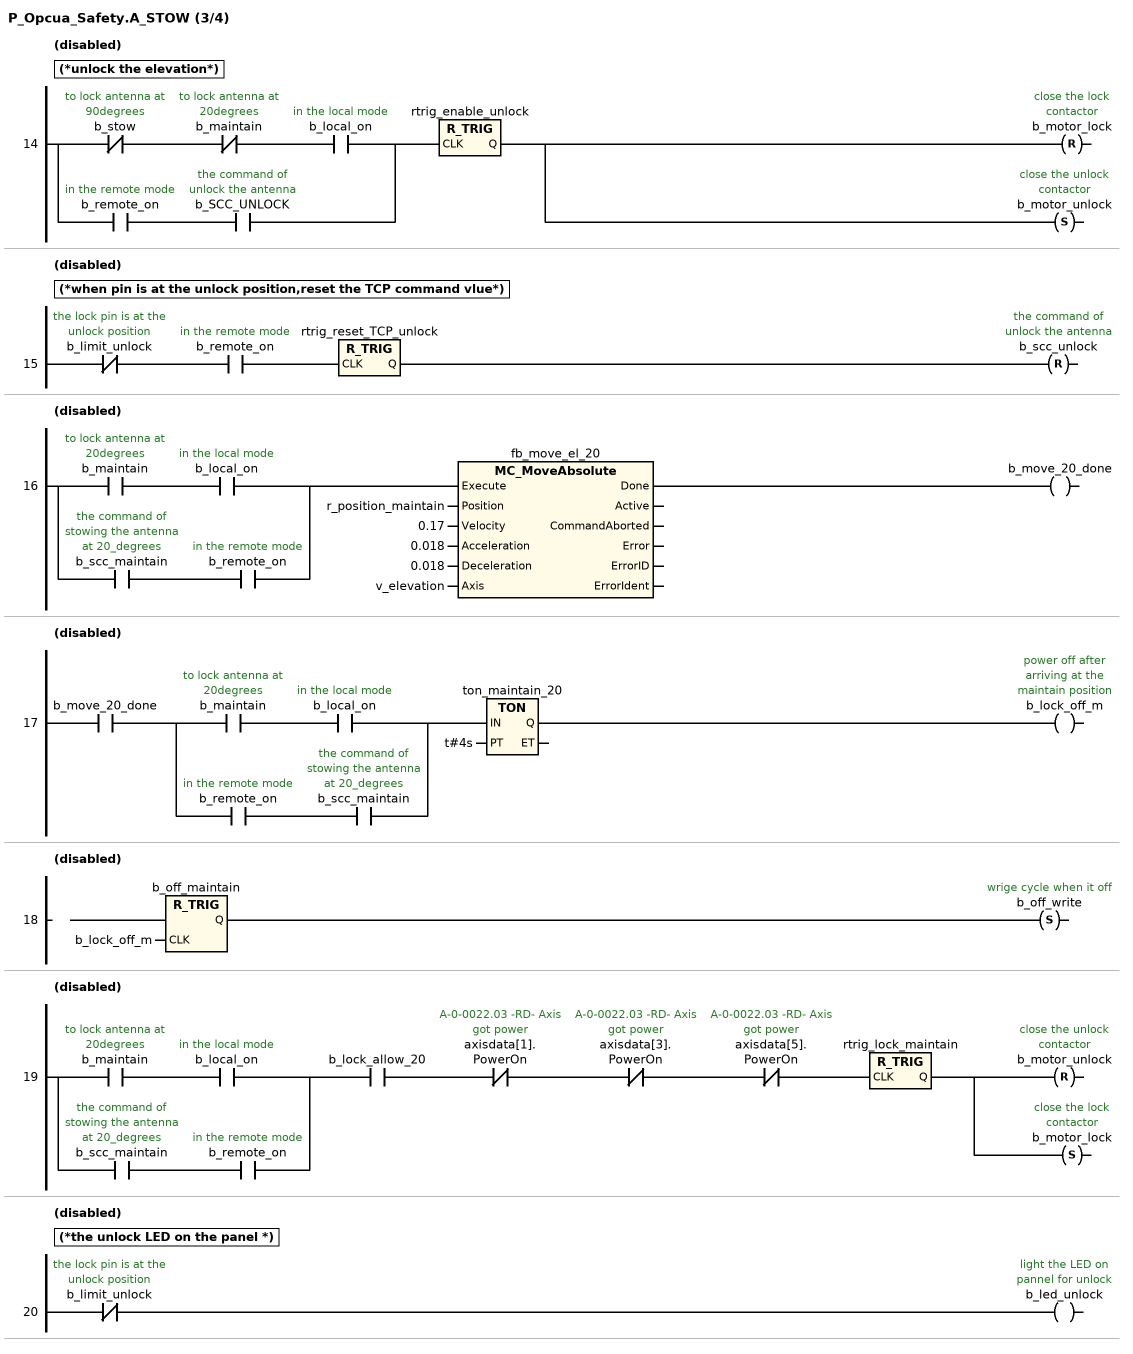
// NETWORK 14 (disabled)
//   b_stow: to lock antenna at 90degrees
//   b_maintain: to lock antenna at 20degrees
//   b_local_on: in the local mode
//   b_remote_on: in the remote mode
//   b_SCC_UNLOCK: the command of unlock the antenna
//   b_motor_lock: close the lock contactor
//   b_motor_unlock: close the unlock contactor
// label: (*unlock the elevation*)
// rtrig_enable_unlock(CLK := NOT b_stow AND NOT b_maintain AND b_local_on OR b_remote_on AND b_SCC_UNLOCK); // R_TRIG
// b_motor_lock R= rtrig_enable_unlock.Q;
// b_motor_unlock S= rtrig_enable_unlock.Q;

// NETWORK 15 (disabled)
//   b_limit_unlock: the lock pin is at the unlock position
//   b_remote_on: in the remote mode
//   b_scc_unlock: the command of unlock the antenna
// label: (*when pin is at the unlock position,reset the TCP command vlue*)
// rtrig_reset_TCP_unlock(CLK := NOT b_limit_unlock AND b_remote_on); // R_TRIG
// b_scc_unlock R= rtrig_reset_TCP_unlock.Q;

// NETWORK 16 (disabled)
//   b_maintain: to lock antenna at 20degrees
//   b_local_on: in the local mode
//   b_scc_maintain: the command of stowing the antenna at 20_degrees
//   b_remote_on: in the remote mode
//   v_elevation: Virtual axis "v_elevation" with axis number 8
// fb_move_el_20(
//     Execute := b_maintain AND b_local_on OR b_scc_maintain AND b_remote_on,
//     Position := r_position_maintain,
//     Velocity := 0.17,
//     Acceleration := 0.018,
//     Deceleration := 0.018,
//     Axis := v_elevation); // MC_MoveAbsolute
// b_move_20_done := fb_move_el_20.Done;

// NETWORK 17 (disabled)
//   b_maintain: to lock antenna at 20degrees
//   b_local_on: in the local mode
//   b_remote_on: in the remote mode
//   b_scc_maintain: the command of stowing the antenna at 20_degrees
//   b_lock_off_m: power off after arriving at the maintain position
// ton_maintain_20(IN := b_move_20_done AND (b_maintain AND b_local_on OR b_remote_on AND b_scc_maintain), PT := t#4s); // TON
// b_lock_off_m := ton_maintain_20.Q;

// NETWORK 18 (disabled)
//   b_lock_off_m: power off after arriving at the maintain position
//   b_off_write: wrige cycle when it off
// b_off_maintain(CLK := b_lock_off_m); // R_TRIG
// b_off_write S= b_off_maintain.Q;

// NETWORK 19 (disabled)
//   b_maintain: to lock antenna at 20degrees
//   b_local_on: in the local mode
//   b_scc_maintain: the command of stowing the antenna at 20_degrees
//   b_remote_on: in the remote mode
//   axisdata[1].PowerOn: A-0-0022.03 -RD- Axis got power
//   axisdata[3].PowerOn: A-0-0022.03 -RD- Axis got power
//   axisdata[5].PowerOn: A-0-0022.03 -RD- Axis got power
//   b_motor_unlock: close the unlock contactor
//   b_motor_lock: close the lock contactor
// rtrig_lock_maintain(CLK := (b_maintain AND b_local_on OR b_scc_maintain AND b_remote_on) AND b_lock_allow_20 AND NOT axisdata[1].PowerOn AND NOT axisdata[3].PowerOn AND NOT axisdata[5].PowerOn); // R_TRIG
// b_motor_unlock R= rtrig_lock_maintain.Q;
// b_motor_lock S= rtrig_lock_maintain.Q;

// NETWORK 20 (disabled)
//   b_limit_unlock: the lock pin is at the unlock position
//   b_led_unlock: light the LED on pannel for unlock
// label: (*the unlock LED on the panel *)
// b_led_unlock := NOT b_limit_unlock;

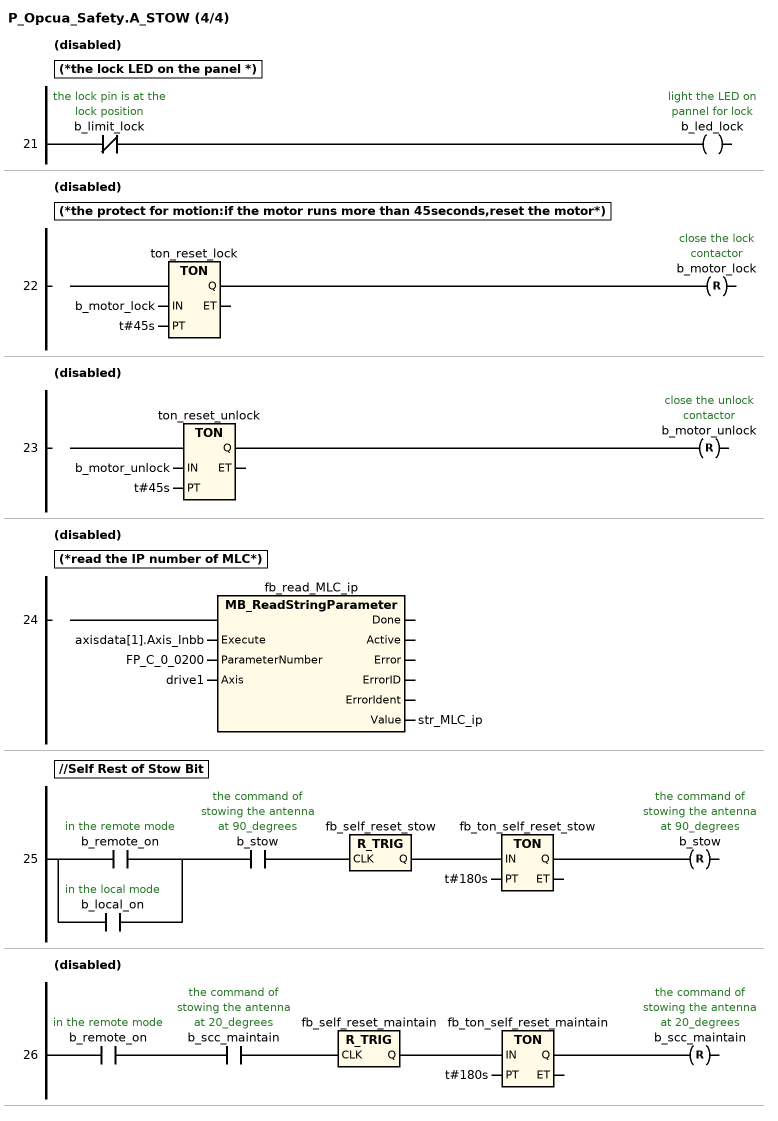
// NETWORK 21 (disabled)
//   b_limit_lock: the lock pin is at the lock position
//   b_led_lock: light the LED on pannel for lock
// label: (*the lock LED on the panel *)
// b_led_lock := NOT b_limit_lock;

// NETWORK 22 (disabled)
//   b_motor_lock: close the lock contactor
// label: (*the protect for motion:if the motor runs more than 45seconds,reset the motor*)
// ton_reset_lock(IN := b_motor_lock, PT := t#45s); // TON
// b_motor_lock R= ton_reset_lock.Q;

// NETWORK 23 (disabled)
//   b_motor_unlock: close the unlock contactor
// ton_reset_unlock(IN := b_motor_unlock, PT := t#45s); // TON
// b_motor_unlock R= ton_reset_unlock.Q;

// NETWORK 24 (disabled)
//   axisdata[1].Axis_Inbb: A-0-0021.13 -RD- Axis is ready for power to the amplifier (bb)
//   FP_C_0_0200: Engineering, IP address
//   drive1: Real axis "Drive1" with axis number 1
//   str_MLC_ip: IP number in MLC
// label: (*read the IP number of MLC*)
// fb_read_MLC_ip(
//     Execute := axisdata[1].Axis_Inbb,
//     ParameterNumber := FP_C_0_0200,
//     Axis := drive1,
//     Value => str_MLC_ip); // MB_ReadStringParameter

// NETWORK 25
//   b_remote_on: in the remote mode
//   b_local_on: in the local mode
//   b_stow: the command of stowing the antenna at 90_degrees
// label: //Self Rest of Stow Bit
fb_self_reset_stow(CLK := (b_remote_on OR b_local_on) AND b_stow); // R_TRIG
fb_ton_self_reset_stow(IN := fb_self_reset_stow.Q, PT := t#180s); // TON
b_stow R= fb_ton_self_reset_stow.Q;

// NETWORK 26 (disabled)
//   b_remote_on: in the remote mode
//   b_scc_maintain: the command of stowing the antenna at 20_degrees
// fb_self_reset_maintain(CLK := b_remote_on AND b_scc_maintain); // R_TRIG
// fb_ton_self_reset_maintain(IN := fb_self_reset_maintain.Q, PT := t#180s); // TON
// b_scc_maintain R= fb_ton_self_reset_maintain.Q;
END_ACTION

ACTION A_Interlock_Estop:
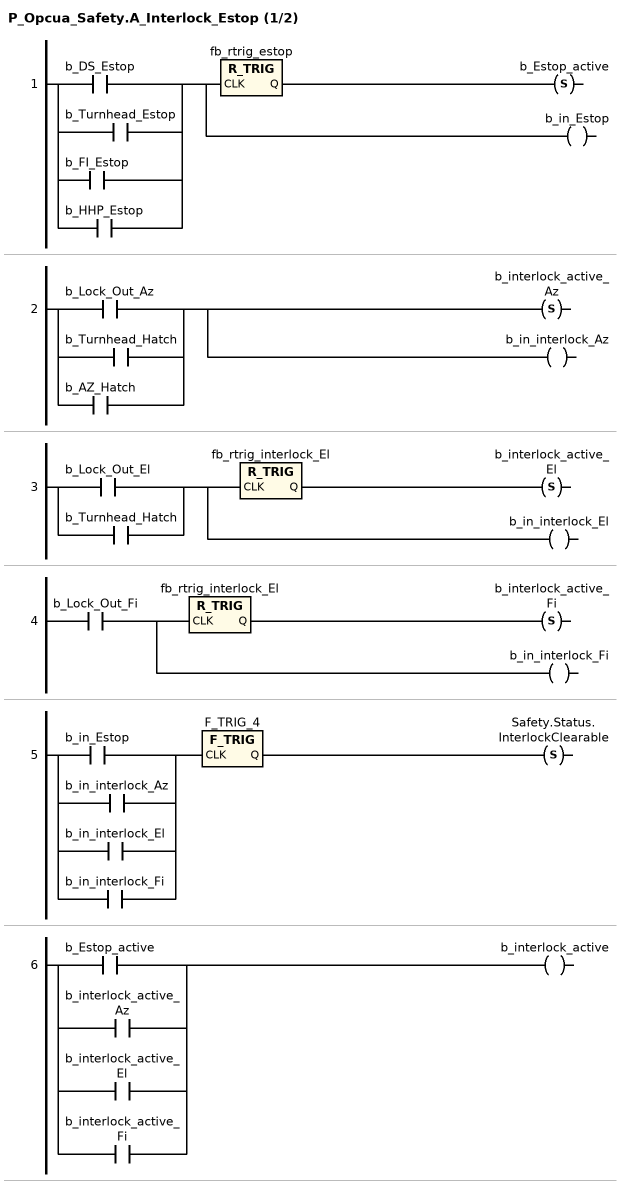
// NETWORK 1
_w3 := b_DS_Estop OR b_Turnhead_Estop OR b_FI_Estop OR b_HHP_Estop;
fb_rtrig_estop(CLK := _w3); // R_TRIG
b_Estop_active S= fb_rtrig_estop.Q;
b_in_Estop := _w3;

// NETWORK 2
_w4 := b_Lock_Out_Az OR b_Turnhead_Hatch OR b_AZ_Hatch;
b_interlock_active_Az S= _w4;
b_in_interlock_Az := _w4;

// NETWORK 3
_w5 := b_Lock_Out_El OR b_Turnhead_Hatch;
fb_rtrig_interlock_El(CLK := _w5); // R_TRIG
b_interlock_active_El S= fb_rtrig_interlock_El.Q;
b_in_interlock_El := _w5;

// NETWORK 4
fb_rtrig_interlock_El(CLK := b_Lock_Out_Fi); // R_TRIG
b_interlock_active_Fi S= fb_rtrig_interlock_El.Q;
b_in_interlock_Fi := b_Lock_Out_Fi;

// NETWORK 5
F_TRIG_4(CLK := b_in_Estop OR b_in_interlock_Az OR b_in_interlock_El OR b_in_interlock_Fi); // F_TRIG
Safety.Status.InterlockClearable S= F_TRIG_4.Q;

// NETWORK 6
b_interlock_active := b_Estop_active OR b_interlock_active_Az OR b_interlock_active_El OR b_interlock_active_Fi;

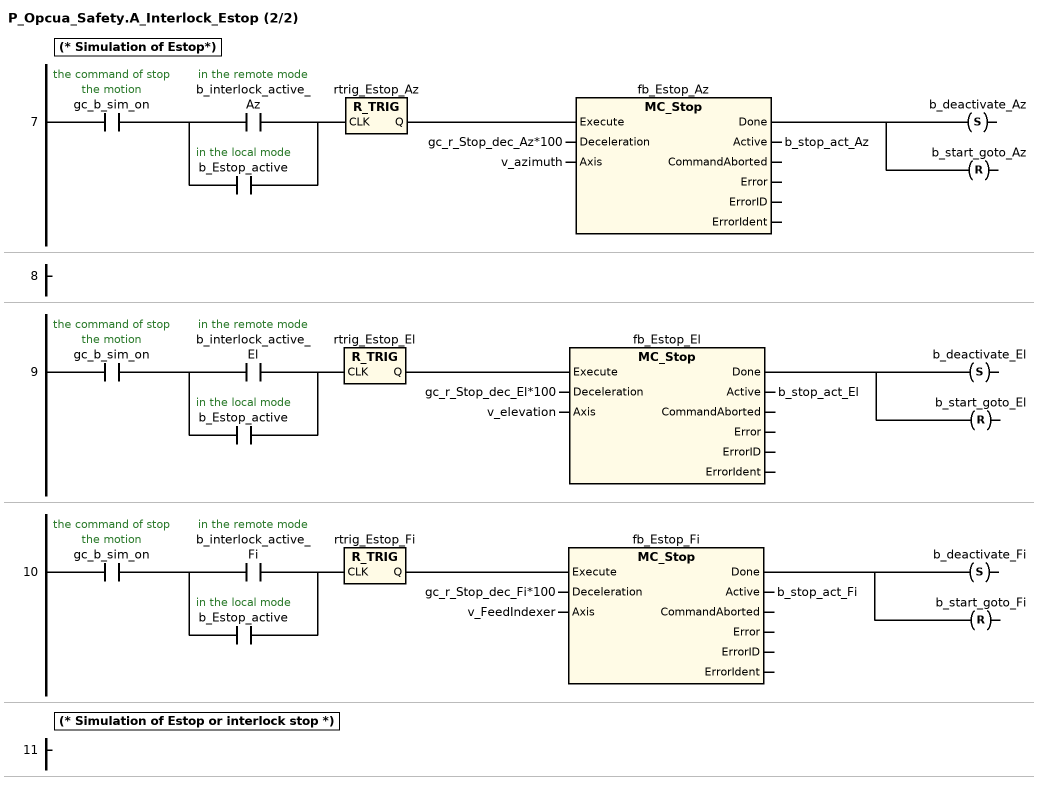
// NETWORK 7
//   gc_b_sim_on: the command of stop the motion
//   b_interlock_active_Az: in the remote mode
//   b_Estop_active: in the local mode
//   v_azimuth: Virtual axis "v_azimuth" with axis number 7
// label: (* Simulation of Estop*)
rtrig_Estop_Az(CLK := gc_b_sim_on AND (b_interlock_active_Az OR b_Estop_active)); // R_TRIG
fb_Estop_Az(
    Execute := rtrig_Estop_Az.Q,
    Deceleration := gc_r_Stop_dec_Az*100,
    Axis := v_azimuth,
    Active => b_stop_act_Az); // MC_Stop
b_deactivate_Az S= fb_Estop_Az.Done;
b_start_goto_Az R= fb_Estop_Az.Done;

// NETWORK 8

// NETWORK 9
//   gc_b_sim_on: the command of stop the motion
//   b_interlock_active_El: in the remote mode
//   b_Estop_active: in the local mode
//   v_elevation: Virtual axis "v_elevation" with axis number 8
rtrig_Estop_El(CLK := gc_b_sim_on AND (b_interlock_active_El OR b_Estop_active)); // R_TRIG
fb_Estop_El(
    Execute := rtrig_Estop_El.Q,
    Deceleration := gc_r_Stop_dec_El*100,
    Axis := v_elevation,
    Active => b_stop_act_El); // MC_Stop
b_deactivate_El S= fb_Estop_El.Done;
b_start_goto_El R= fb_Estop_El.Done;

// NETWORK 10
//   gc_b_sim_on: the command of stop the motion
//   b_interlock_active_Fi: in the remote mode
//   b_Estop_active: in the local mode
//   v_FeedIndexer: Virtual axis "v_polarization" with axis number 9
rtrig_Estop_Fi(CLK := gc_b_sim_on AND (b_interlock_active_Fi OR b_Estop_active)); // R_TRIG
fb_Estop_Fi(
    Execute := rtrig_Estop_Fi.Q,
    Deceleration := gc_r_Stop_dec_Fi*100,
    Axis := v_FeedIndexer,
    Active => b_stop_act_Fi); // MC_Stop
b_deactivate_Fi S= fb_Estop_Fi.Done;
b_start_goto_Fi R= fb_Estop_Fi.Done;

// NETWORK 11
// label: (* Simulation of Estop or interlock stop *)
END_ACTION

END_PROGRAM

// IndraMotionMlc1/Application/POUs/OPCUA/OPCUA_Node/P_Opcua_CommandArbiter
PROGRAM P_Opcua_CommandArbiter
VAR
	cmds: CmdResponseType;
END_VAR

CommandArbiter();
//CommandArbiter.Status.DscCmdAuthority;


(* if hhp connected then 
    CommandArbiter.DscCmdAuthority:= HHP;
	End *)

END_PROGRAM

// IndraMotionMlc1/Application/POUs/OPCUA/OPCUA_Node/P_Opcua_Time_cds
PROGRAM P_Opcua_Time_cds
VAR
	IL_SysTime64_0: IL_SysTime64;
	Current_time: SYS_TIME64;
	UnixSeconds: Lreal;
	i_num_quarter_test: DINT;
	current_time_pos_test: LREAL;
	lr_MJD_Test: LREAL;
	
	dummy: Lreal;
	dummy2: Bool;
END_VAR

Time_cds();

P_Opcua_Time_cds.Get_Time();
//Time_cds.Status.TAIOffset:=Current_time.HighValue*65536+Current_time.LowValue;
//Calculate TAI offset 
//Time_cds.Status.TAIOffset:=Current_time.HighValue*65536+Current_time.LowValue;
//Time_cds.Status.TAIOffset:=((Current_time.HighValue+4294967295)/1000000+ Current_time.LowValue/1000000);
UnixSeconds:=(TO_LREAL(Current_time.HighValue)*4294967295+TO_LREAL(Current_time.LowValue))/1000000; //UTC 
//Time_cds.Status.TAIOffset:=UnixSeconds-UnixToSKAEpoch-(Time_cds.Status.LeapSecPTP-Time_cds.Status.UTCtoSkaoEpochSec);

lr_MJD_Test:= UnixSeconds/86400+40587;

 // This should be the TAI offset after the SKAO epoch. The time from the Time Virtual axis.
//Time_cds.Status.DscTimeSyncSource:=Source_Timesync;

Time_cds.Status.LeapSecPTP:=LeapSecPTP;   
IF Source_Timesync = DscTimeSyncSourceType.PTP THEN
	Time_cds.Status.TimeSourceAddrNTP:=IP_Adress_PTP;
ELSIF Source_Timesync = DscTimeSyncSourceType.NTP THEN
	Time_cds.Status.TimeSourceAddrNTP:=IP_Adress_NTP;
ELSE
	Time_cds.Status.TimeSourceAddrNTP:=str_MLC_ip;
END_IF

IF Source_Timesync = DscTimeSyncSourceType.PTP THEN
	Time_cds.Status.TimeSynced:=b_M_time_done;
	b_no_SetDateTime:=FALSE;
ELSIF Source_Timesync = DscTimeSyncSourceType.NTP THEN
	//Time_cds.Status.TimeSynced:=b_M_time_done;
	b_no_SetDateTime:=FALSE;
ELSE
	
    Time_cds.Status.TimeSynced:=b_M_time_done;
	// need to use system time to calculate MJD
	b_no_SetDateTime:=TRUE;
	
	di_MJD_day := LREAL_TO_DINT(TRUNC(UnixSeconds/86400+40587));
	i_num_quarter:=TRUNC((UnixSeconds-DINT_TO_LREAL(TRUNC(UnixSeconds/86400)*86400))/360);
	current_time_pos_test:=UnixSeconds-DINT_TO_LREAL(TRUNC(UnixSeconds/86400)*86400)-i_num_quarter*360;
	dummy:=P_UDP_To_NTP.current_time_pos-current_time_pos_test;
	dummy2:=(ABS(dummy)>=0.10);
	IF (ABS(dummy)>=0.10 AND NOT(b_track_on)) THEN
		P_UDP_To_NTP.current_time_pos:=current_time_pos_test;
	   	P_UDP_To_NTP.b_NTP_set_up:=TRUE;
	ELSE 
		P_UDP_To_NTP.b_NTP_set_up:=FALSE;	
	
	END_IF
	
	
	
END_IF

ACTION Get_Time:
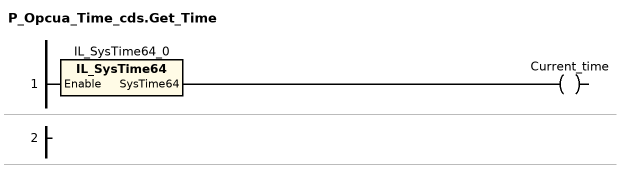
// NETWORK 1
IL_SysTime64_0(Enable := TRUE); // IL_SysTime64
Current_time := IL_SysTime64_0.SysTime64;

// NETWORK 2
END_ACTION

END_PROGRAM

// IndraMotionMlc1/Application/POUs/OPCUA/OPCUA_Node/P_Opcua_Management
PROGRAM P_Opcua_Management
VAR
	R_total_distance_AZ_old:LREAL;
	R_total_distance_EL_deg_old:LREAL;
	R_total_distance_EL_m_old:LREAL;
	R_total_distance_FI_old:LREAL;
	count_i:UINT;
	(*<<<<<<<<<<<<<<<<<<<<<<<<<<<<<<<<<<<< Stop >>>>>>>>>>>>>>>>>>>>>>>>>>>>>*)
	b_stop_Az_done: BOOL;
	b_stop_El_done: BOOL;
	b_stop_Fi_done: BOOL;
	fb_stop_Az: MC_Stop;
	fb_stop_El: MC_Stop;
	fb_stop_Fi: MC_Stop;
	rtrig_stop_Az: R_TRIG;
	rtrig_stop_El: R_TRIG;
	rtrig_stop_Fi: R_TRIG;
	rtrig_stop_stow: R_TRIG;
	rtrig_reset_stop: R_TRIG;
	
	(*<<<<<<<<<<<<<<<<<<<<<<<<<<<<<<<<<<<< Goto >>>>>>>>>>>>>>>>>>>>>>>>>>>>>*)
	// Az
	
	b_goto_done_Az: BOOL;
	b_active_Az:     BOOL;
	b_moving_Az: BOOL;
	fb_goto_Az: MC_MoveRelative;
	fb_start_goto_Az: R_Trig;
	fb_goto_done_Az : R_Trig;
	
	// El
	
	b_goto_done_El: BOOL;
	b_active_El:     BOOL;
	b_moving_El: BOOL;
	fb_goto_El: MC_MoveRelative;
	fb_start_goto_El: R_Trig;
	fb_goto_done_El : R_Trig;
	//Fi
	b_goto_done_Fi: BOOL;
	b_active_Fi:     BOOL;
	b_moving_Fi: BOOL;
	fb_goto_Fi: MC_MoveRelative;
	fb_start_goto_Fi: R_Trig;
	fb_goto_done_Fi : R_Trig;
	
(*<<<<<<<<<<<<<<<<<<<<<<<<<<<<<<<<<<<<<<<<<<<<<<<<<<<power>>>>>>>>>>>>>>>>>>>>>>>>>>>>>>>>>>>>*)
	ton_pow_off_Az: TON;
	ton_pow_off_El: TON;
	ton_pow_off_Fi: TON;
	rtrig_power_Az: R_TRIG;
	rtrig_power_El: R_TRIG;
	rtrig_power_Fi: R_TRIG;
	fb_ton_El: TON;
	fb_ton_Fi: TON;
	rtrig_off_Az: R_TRIG;
	rtrig_off_El: R_TRIG;
	rtrig_off_Fi: R_TRIG;
	rtrig_power_power: R_TRIG;
	b_pwr_on:BOOL;
	b_pwr_off: BOOL;
	b_clear_off_done_Az1: BOOL;
	b_clear_off_done_Az2: BOOL;
	b_clear_off_done_El: BOOL;
	b_clear_off_done_Fi1: BOOL;
	b_clear_off_done_Fi2: BOOL;
	
	FB_clear_error_off_Az1:MB_WriteParameter;
	FB_clear_error_off_Az2:MB_WriteParameter;
	FB_clear_error_off_El:MB_WriteParameter;
	FB_clear_error_off_Fi1:MB_WriteParameter;
	FB_clear_error_off_Fi2:MB_WriteParameter;
	rtrig_err: R_TRIG;
	rtrig_clear_done: R_TRIG;
	fb_ton_stow: TON;
	
	fb_rtrig_stow_deactivate1: R_TRIG;
	fb_rtrig_stow_deactivate: R_TRIG;
	b_execute_goto_Az: BOOL;
	TON_0: TON;
	R_TRIG_0: R_TRIG;
	R_TRIG_1: R_TRIG;
	TON_1: TON;
END_VAR


(***********Management.DscState***********)
IF azimuth.Status.AxisState=axisstatetype.StartUp OR elevation.Status.AxisState=axisstatetype.StartUp THEN
	Management.Status.DscState:=DscstateType.StartUp;
END_IF

IF azimuth.Status.AxisState=axisstatetype.Standby AND elevation.Status.AxisState=axisstatetype.Standby THEN
	Management.Status.DscState:=DscstateType.Standby;
END_IF

IF azimuth.Status.AxisState=axisstatetype.Activating OR elevation.Status.AxisState=axisstatetype.Activating THEN
	Management.Status.DscState:=DscstateType.Activating;
END_IF

IF azimuth.Status.AxisState=axisstatetype.Deactivating OR elevation.Status.AxisState=axisstatetype.Deactivating THEN
	Management.Status.DscState:=DscstateType.Deactivating;
END_IF

IF azimuth.Status.AxisState=axisstatetype.Standstill OR elevation.Status.AxisState=axisstatetype.Standstill THEN
	Management.Status.DscState:=DscstateType.Standstill;
END_IF

IF azimuth.Status.AxisState=axisstatetype.Stopping OR elevation.Status.AxisState=axisstatetype.Stopping THEN
	Management.Status.DscState:=DscstateType.stopping;
END_IF

IF azimuth.Status.AxisState=axisstatetype.Jog OR elevation.Status.AxisState=axisstatetype.Jog THEN
	Management.Status.DscState:=DscstateType.Jog;
END_IF

IF azimuth.Status.AxisState=axisstatetype.Slew OR elevation.Status.AxisState=axisstatetype.Slew THEN //capitalise S in slew
	Management.Status.DscState:=DscstateType.slew;
END_IF

IF azimuth.Status.AxisState=axisstatetype.Track AND elevation.Status.AxisState=axisstatetype.Track THEN
	Management.Status.DscState:=DscstateType.Track;
END_IF

IF azimuth.Status.AxisState=axisstatetype.Stowed THEN
	Management.Status.DscState:=DscstateType.Stowed;
END_IF
IF azimuth.Status.AxisState=axisstatetype.Locked OR elevation.Status.AxisState=axisstatetype.Locked THEN
	Management.Status.DscState:=DscstateType.Locked;
END_IF

IF azimuth.Status.AxisState=axisstatetype.Locked_Stowed OR elevation.Status.AxisState=axisstatetype.Locked_Stowed THEN
	Management.Status.DscState:=DscstateType.Locked_Stowed;
END_IF

// This one isn't going to work 
IF b_stow_pin_limit_lock AND (azimuth.Status.AxisState=axisstatetype.Locked OR elevation.Status.AxisState=axisstatetype.Locked) THEN     // Need to check Errors and interlocks to go into locked
	Management.Status.DscState:=DscstateType.Locked_Stowed;
END_IF

(*IF b_in_Estop THEN
	Management.Status.DscState:=DscstateType.Locked;  //Axis also need to go into locked state
END_IF
*)


// Work out where FiPOS is 
IF b_goto_done_Fi THEN 
	IF r_pos_fi_v < gc_r_band_optical+gc_r_band_tolerance AND r_pos_fi_v > gc_r_band_optical-gc_r_band_tolerance THEN 
		Management.Status.FiPos:= bandtype.Optical;
	ELSIF
		r_pos_fi_v < gc_r_band_1+gc_r_band_tolerance AND r_pos_fi_v > gc_r_band_1-gc_r_band_tolerance THEN 
		Management.Status.FiPos:= bandtype.Band_1;
	ELSIF
		r_pos_fi_v < gc_r_band_2+gc_r_band_tolerance AND r_pos_fi_v > gc_r_band_2-gc_r_band_tolerance THEN 
		Management.Status.FiPos:= bandtype.Band_2;
	ELSIF
		r_pos_fi_v < gc_r_band_3+gc_r_band_tolerance AND r_pos_fi_v > gc_r_band_3-gc_r_band_tolerance THEN 
		Management.Status.FiPos:= bandtype.Band_3;
	ELSIF
		r_pos_fi_v < gc_r_band_4+gc_r_band_tolerance AND r_pos_fi_v > gc_r_band_4-gc_r_band_tolerance THEN 
		Management.Status.FiPos:= bandtype.Band_4;
	ELSIF
		r_pos_fi_v < gc_r_band_5a+gc_r_band_tolerance AND r_pos_fi_v > gc_r_band_5a-gc_r_band_tolerance THEN 
		Management.Status.FiPos:= bandtype.Band_5a;
	ELSIF
		r_pos_fi_v < gc_r_band_5b+gc_r_band_tolerance AND r_pos_fi_v > gc_r_band_5b-gc_r_band_tolerance THEN 
		Management.Status.FiPos:= bandtype.Band_5b;
	ELSIF
		r_pos_fi_v < gc_r_band_6+gc_r_band_tolerance AND r_pos_fi_v > gc_r_band_6-gc_r_band_tolerance THEN 
		Management.Status.FiPos:= bandtype.Band_6;
	ELSE
		Management.Status.FiPos:= bandtype.Unknown;
	END_IF

END_IF


//Management.Status.FiPos:=Current_FIPos; // this needs to be of band type 
Management.Status.HHP_Cncted:=b_HHP_Connected;
Management.Status.HHP_Az:=b_HHP_AZ;
Management.Status.HHP_El:=b_HHP_EL;
IF b_HHP_AZ = FALSE AND b_HHP_EL= FALSE THEN
	Management.Status.HHP_Fi:=TRUE;
ELSE
	Management.Status.HHP_Fi:=FALSE;
END_IF
IF b_HHP_move_cw_slow OR b_HHP_move_cw_fast THEN
	Management.Status.HHP_Dir_Plus	:= TRUE;
ELSE
	Management.Status.HHP_Dir_Plus	:= FALSE;
END_IF
IF b_HHP_move_ccw_slow OR b_HHP_move_ccw_fast THEN
	Management.Status.HHP_Dir_Minus:= TRUE;
ELSE
	Management.Status.HHP_Dir_Minus:= FALSE;
END_IF

(*********NamePlate**********)
Management.NamePlate.RunHours:=r_operation_hour;

count_i:=count_i+1;
IF count_i = 5 THEN
	R_total_distance_AZ:=ABS(r_pos_az-R_total_distance_AZ_old)+R_total_distance_AZ;
	R_total_distance_AZ_old:=r_pos_az;
	R_total_distance_EL_deg:=ABS(r_pos_el-R_total_distance_el_deg_old)+R_total_distance_el_deg;
	R_total_distance_EL_m:=R_total_distance_EL_deg/K_gear_ratio;
	R_total_distance_el_deg_old:=r_pos_el;
	R_total_distance_FI:=ABS(r_pos_FI-R_total_distance_FI_old)+R_total_distance_FI;
	R_total_distance_FI_old:=r_pos_FI;
	count_i:=0;
END_IF

Management.NamePlate.TotalDist_Az:=R_total_distance_AZ;
Management.NamePlate.TotalDist_El_deg:=R_total_distance_EL_deg;
Management.NamePlate.TotalDist_El_m:=R_total_distance_EL_m;
Management.NamePlate.TotalDist_Fi:=R_total_distance_FI;

(*********TempHumidStatus**********)
Management.TempHumidStatus.HumidDriveCab:=LREAL_TO_REAL(HumidDriveCab);
Management.TempHumidStatus.TempDriveCab:=LREAL_TO_REAL(TempDriveCab);
Management.TempHumidStatus.HumidPSC_Inlet:=LREAL_TO_REAL(HumidPSC_Inlet);
Management.TempHumidStatus.TempPSC_Inlet:=LREAL_TO_REAL(TempPSC_Inlet);
Management.TempHumidStatus.HumidPSC_Outlet:=LREAL_TO_REAL(HumidPSC_Outlet);
Management.TempHumidStatus.TempPSC_Outlet:=LREAL_TO_REAL(TempPSC_Outlet);
Management.TempHumidStatus.TempEMISC_Outlet:=LREAL_TO_REAL(TempEMISC_Outlet);

(*********PowerStatus**********)
Management.PowerStatus.cbEMISC:=b_PSC_PD_EMISC_Breaker_on;
Management.PowerStatus.cbFan_PSC:=b_PSC_PD_FAN_Breaker_on;
Management.PowerStatus.cbPSC_Spare:=b_PSC_PD_spare;
Management.PowerStatus.cbHe_Comp:=b_MAIN_PD_Compressor_breaker_on;
Management.PowerStatus.cbPDU_Fi:=b_MAIN_PD_FI_Breaker_on;
Management.PowerStatus.cbPED_Spare:=b_MAIN_PD_spare;
Management.PowerStatus.ActPwrCnsm:= 0; // Needs to be updated with real number
Management.PowerStatus.CurrentPh1:= LREAL_TO_REAL(CurrentPh1);
Management.PowerStatus.CurrentPh2:=LREAL_TO_REAL(CurrentPh2);
Management.PowerStatus.CurrentPh3:=LREAL_TO_REAL(CurrentPh3);
Management.PowerStatus.FrequencyPh1:=LREAL_TO_REAL(FrequencyPh1);
Management.PowerStatus.FrequencyPh2:=LREAL_TO_REAL(FrequencyPh2);
Management.PowerStatus.FrequencyPh3:=LREAL_TO_REAL(FrequencyPh3);
Management.PowerStatus.VoltagePh1:=LREAL_TO_REAL(VoltagePh1);
Management.PowerStatus.VoltagePh2:=LREAL_TO_REAL(VoltagePh2);
Management.PowerStatus.VoltagePh3:=LREAL_TO_REAL(VoltagePh3);
Management.PowerStatus.PowerFactor:=LREAL_TO_REAL(PowerFactor);
//Management.PowerStatus.LowPowerActive:=0;  

(*********ErrorStatus**********)

//Management.ErrorStatus.errAuthLost:=0;
Management.ErrorStatus.errAzimuth:=(axisdata[1].Axis_Error OR axisdata[2].Axis_Error);  
Management.ErrorStatus.errElevation:=(axisdata[3].Axis_Error);  
Management.ErrorStatus.errFeedindexer:=(axisdata[4].Axis_Error OR axisdata[5].Axis_Error); 
Management.ErrorStatus.errPoint:=0;
IF safety.Status.SafetyState=0 THEN
	Management.ErrorStatus.errSafety:=0;
ELSE
	Management.ErrorStatus.errSafety:=1;
END_IF
Management.ErrorStatus.errTime:=axisdata[10].Axis_Error;
Management.ErrorStatus.errCmd:=Command_Arbiter_error;
Management.ErrorStatus.errTrack:=(NOT(tracking.Status.tr_initOk) AND b_track_on);
Management.ErrorStatus.errStwPin:=NOT((b_stow_pin_limit_lock XOR b_stow_pin_limit_unlock)XOR(b_stow_pin_retract XOR b_stow_pin_deploy));
IF status_code1 = 'F8070' OR status_code2 = 'F8070' OR status_code3 = 'F8070' OR status_code4 = 'F8070' OR status_code5 = 'F8070' THEN
	Management.ErrorStatus.errPwr24VDC:=1;
ELSE
	Management.ErrorStatus.errPwr24VDC:=0;
END_IF
IF status_code1 = 'F2802' OR status_code2 = 'F2802' OR status_code3 = 'F2802' OR status_code4 = 'F2802' OR status_code5 = 'F2802' THEN
	Management.ErrorStatus.errPwr400VAC:=1;
ELSE
	Management.ErrorStatus.errPwr400VAC:=0;
END_IF
IF status_code1 = 'F2802' OR status_code2 = 'F2802' OR status_code3 = 'F2802' OR status_code4 = 'F2802' OR status_code5 = 'F2802' THEN
	Management.ErrorStatus.errPwr400VAC:=1;
ELSE
	Management.ErrorStatus.errPwr400VAC:=0;
END_IF
IF status_code1 = 'F8091' OR status_code2 = 'F8091' OR status_code3 = 'F8091' OR status_code4 = 'F8091' OR status_code5 = 'F8091' THEN
	Management.ErrorStatus.errPwr400VAC:=1;
ELSE
	Management.ErrorStatus.errPwr400VAC:=0;
END_IF
//	Management.ErrorStatus.errPwrMeterComms:=0;
//	Management.ErrorStatus.errTiltOneComms:=0;
//	Management.ErrorStatus.errTiltOneIoUnit:=0;
//	Management.ErrorStatus.errTiltTwoComms:=0;
//	Management.ErrorStatus.errTiltTwoIoUnit:=0;

Management.ErrorStatus.errGeneral:=(Management.ErrorStatus.errAzimuth OR Management.ErrorStatus.errElevation OR Management.ErrorStatus.errFeedindexer OR Management.ErrorStatus.errSafety OR Management.ErrorStatus.errTime OR Management.ErrorStatus.errTrack OR Management.ErrorStatus.errPoint);
Management.ErrorStatus.errMngmnt:=Management.ErrorStatus.errGeneral;

(*********WarningStatus**********)
//IF gc_b_sim_on = 0 THEN 
	Management.WarningStatus.waAzimuth:=(axisdata[1].Axis_Warning OR axisdata[2].Axis_Warning);
    Management.WarningStatus.waElevation:=(axisdata[3].Axis_Warning);
    Management.WarningStatus.waFeedindexer:=(axisdata[4].Axis_Warning OR axisdata[5].Axis_Warning);
//ELSIF gc_b_sim_on =1 THEN
//	Management.WarningStatus.waAzimuth:=(

Management.WarningStatus.waCmd:=0;
Management.WarningStatus.waPoint:=0;
Management.WarningStatus.waSafety:=0;
Management.WarningStatus.waStwPin:=0;
Management.WarningStatus.waPoint:=0;
Management.WarningStatus.waTime:=0;
Management.WarningStatus.waTrack:=0;
Management.WarningStatus.waDoorDrive:=b_DriveCabinetDoor_Estop;
Management.WarningStatus.waDoorEMISC:=b_EMISCDoor_Estop;
Management.WarningStatus.waDoorPED:=b_DSDoor_Estop;
Management.WarningStatus.waDoorPSC:=b_PSCDoor_Estop;
Management.WarningStatus.waHatchPscRoof:=0;
Management.WarningStatus.waHatchAzBearing:=b_AZ_Hatch;
Management.WarningStatus.waHornOn:=b_Horn;
//Management.WarningStatus.waOverTempDrive
//Management.WarningStatus.waOverTempEMISC
//Management.WarningStatus.waDoorPED
//Management.WarningStatus.waDoorPSC
Management.WarningStatus.waSafe2ApproachLight:=0;

// Power mode control 
// Need to limit velocity and acceleration to keep the power below the limit 


// Run Ladder logic
P_Opcua_Management.A_CLR_ERR();
P_Opcua_Management.A_STOP();
P_Opcua_Management.A_GOTO();

ACTION A_STOP:
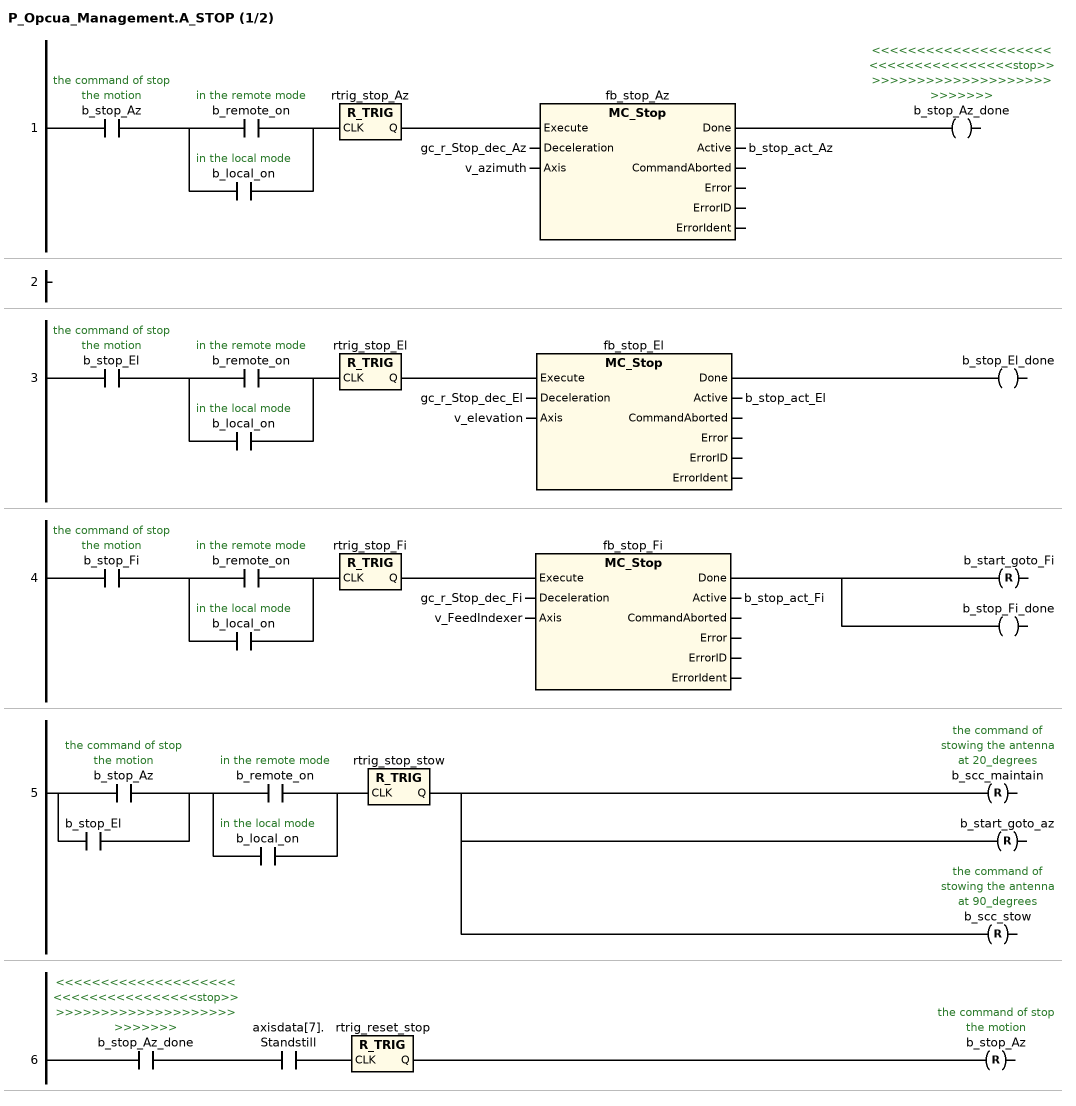
// NETWORK 1
//   b_stop_Az: the command of stop the motion
//   b_remote_on: in the remote mode
//   b_local_on: in the local mode
//   v_azimuth: Virtual axis "v_azimuth" with axis number 7
//   b_stop_Az_done: <<<<<<<<<<<<<<<<<<<<<<<<<<<<<<<<<<<<stop>>>>>>>>>>>>>>>>>>>>>>>>>>>>>
rtrig_stop_Az(CLK := b_stop_Az AND (b_remote_on OR b_local_on)); // R_TRIG
fb_stop_Az(
    Execute := rtrig_stop_Az.Q,
    Deceleration := gc_r_Stop_dec_Az,
    Axis := v_azimuth,
    Active => b_stop_act_Az); // MC_Stop
b_stop_Az_done := fb_stop_Az.Done;

// NETWORK 2

// NETWORK 3
//   b_stop_El: the command of stop the motion
//   b_remote_on: in the remote mode
//   b_local_on: in the local mode
//   v_elevation: Virtual axis "v_elevation" with axis number 8
rtrig_stop_El(CLK := b_stop_El AND (b_remote_on OR b_local_on)); // R_TRIG
fb_stop_El(
    Execute := rtrig_stop_El.Q,
    Deceleration := gc_r_Stop_dec_El,
    Axis := v_elevation,
    Active => b_stop_act_El); // MC_Stop
b_stop_El_done := fb_stop_El.Done;

// NETWORK 4
//   b_stop_Fi: the command of stop the motion
//   b_remote_on: in the remote mode
//   b_local_on: in the local mode
//   v_FeedIndexer: Virtual axis "v_polarization" with axis number 9
rtrig_stop_Fi(CLK := b_stop_Fi AND (b_remote_on OR b_local_on)); // R_TRIG
fb_stop_Fi(
    Execute := rtrig_stop_Fi.Q,
    Deceleration := gc_r_Stop_dec_Fi,
    Axis := v_FeedIndexer,
    Active => b_stop_act_Fi); // MC_Stop
b_start_goto_Fi R= fb_stop_Fi.Done;
b_stop_Fi_done := fb_stop_Fi.Done;

// NETWORK 5
//   b_stop_Az: the command of stop the motion
//   b_remote_on: in the remote mode
//   b_local_on: in the local mode
//   b_scc_maintain: the command of stowing the antenna at 20_degrees
//   b_scc_stow: the command of stowing the antenna at 90_degrees
rtrig_stop_stow(CLK := (b_stop_Az OR b_stop_El) AND (b_remote_on OR b_local_on)); // R_TRIG
b_scc_maintain R= rtrig_stop_stow.Q;
b_start_goto_az R= rtrig_stop_stow.Q;
b_scc_stow R= rtrig_stop_stow.Q;

// NETWORK 6
//   b_stop_Az_done: <<<<<<<<<<<<<<<<<<<<<<<<<<<<<<<<<<<<stop>>>>>>>>>>>>>>>>>>>>>>>>>>>>>
//   b_stop_Az: the command of stop the motion
rtrig_reset_stop(CLK := b_stop_Az_done AND axisdata[7].Standstill); // R_TRIG
b_stop_Az R= rtrig_reset_stop.Q;

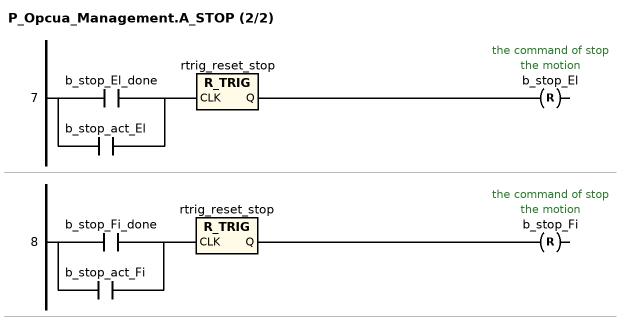
// NETWORK 7
//   b_stop_El: the command of stop the motion
rtrig_reset_stop(CLK := b_stop_El_done OR b_stop_act_El); // R_TRIG
b_stop_El R= rtrig_reset_stop.Q;

// NETWORK 8
//   b_stop_Fi: the command of stop the motion
rtrig_reset_stop(CLK := b_stop_Fi_done OR b_stop_act_Fi); // R_TRIG
b_stop_Fi R= rtrig_reset_stop.Q;
END_ACTION

ACTION A_GOTO:
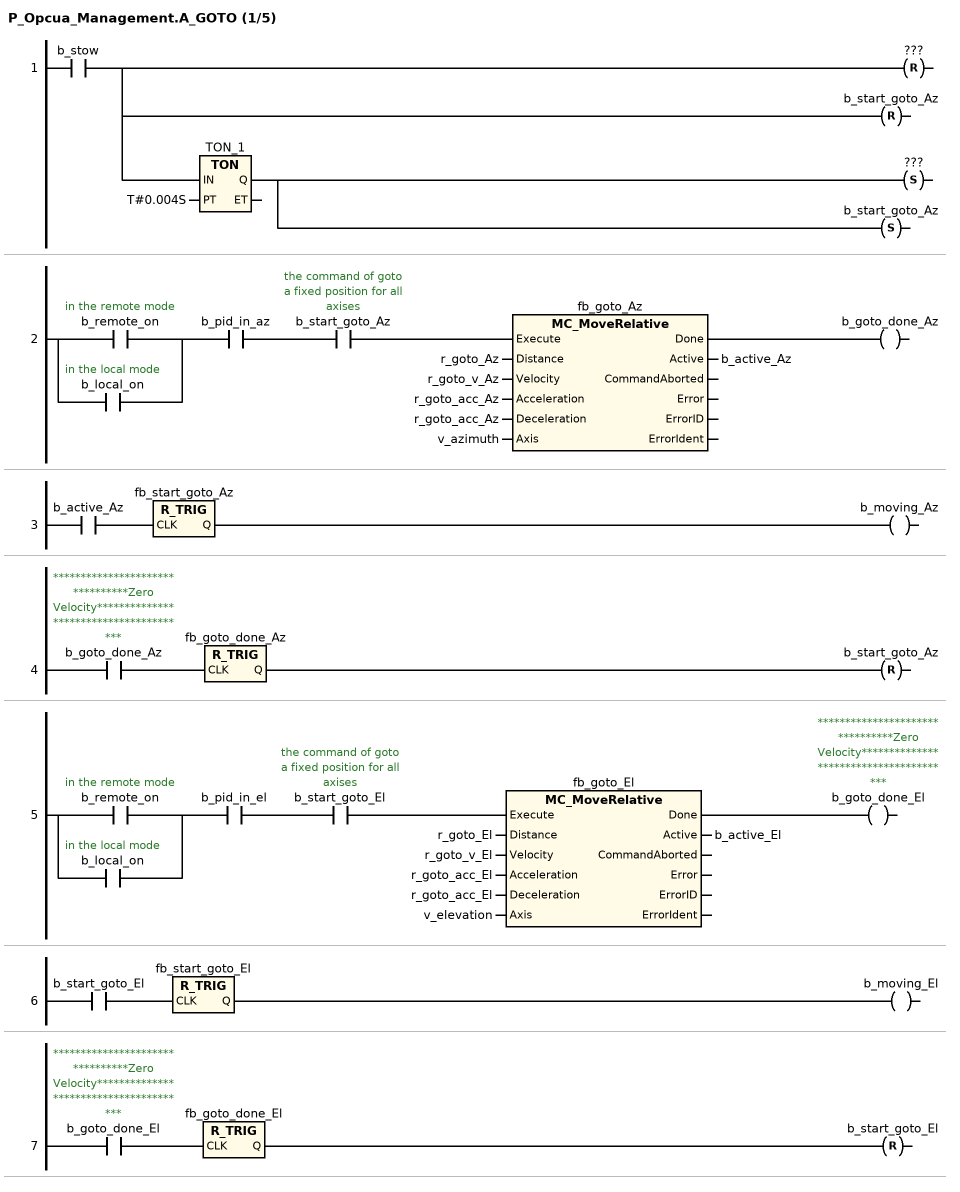
// NETWORK 1
??? R= b_stow;
b_start_goto_Az R= b_stow;
TON_1(IN := b_stow, PT := T#0.004S); // TON
??? S= TON_1.Q;
b_start_goto_Az S= TON_1.Q;

// NETWORK 2
//   b_remote_on: in the remote mode
//   b_local_on: in the local mode
//   b_start_goto_Az: the command of goto a fixed position for all axises
//   r_goto_Az: actual value of goto
//   v_azimuth: Virtual axis "v_azimuth" with axis number 7
fb_goto_Az(
    Execute := (b_remote_on OR b_local_on) AND b_pid_in_az AND b_start_goto_Az,
    Distance := r_goto_Az,
    Velocity := r_goto_v_Az,
    Acceleration := r_goto_acc_Az,
    Deceleration := r_goto_acc_Az,
    Axis := v_azimuth,
    Active => b_active_Az); // MC_MoveRelative
b_goto_done_Az := fb_goto_Az.Done;

// NETWORK 3
fb_start_goto_Az(CLK := b_active_Az); // R_TRIG
b_moving_Az := fb_start_goto_Az.Q;

// NETWORK 4
//   b_goto_done_Az: ********************************Zero Velocity***************************************
fb_goto_done_Az(CLK := b_goto_done_Az); // R_TRIG
b_start_goto_Az R= fb_goto_done_Az.Q;

// NETWORK 5
//   b_remote_on: in the remote mode
//   b_local_on: in the local mode
//   b_start_goto_El: the command of goto a fixed position for all axises
//   r_goto_El: actual value of goto
//   v_elevation: Virtual axis "v_azimuth" with axis number 7
//   b_goto_done_El: ********************************Zero Velocity***************************************
fb_goto_El(
    Execute := (b_remote_on OR b_local_on) AND b_pid_in_el AND b_start_goto_El,
    Distance := r_goto_El,
    Velocity := r_goto_v_El,
    Acceleration := r_goto_acc_El,
    Deceleration := r_goto_acc_El,
    Axis := v_elevation,
    Active => b_active_El); // MC_MoveRelative
b_goto_done_El := fb_goto_El.Done;

// NETWORK 6
fb_start_goto_El(CLK := b_start_goto_El); // R_TRIG
b_moving_El := fb_start_goto_El.Q;

// NETWORK 7
//   b_goto_done_El: ********************************Zero Velocity***************************************
fb_goto_done_El(CLK := b_goto_done_El); // R_TRIG
b_start_goto_El R= fb_goto_done_El.Q;

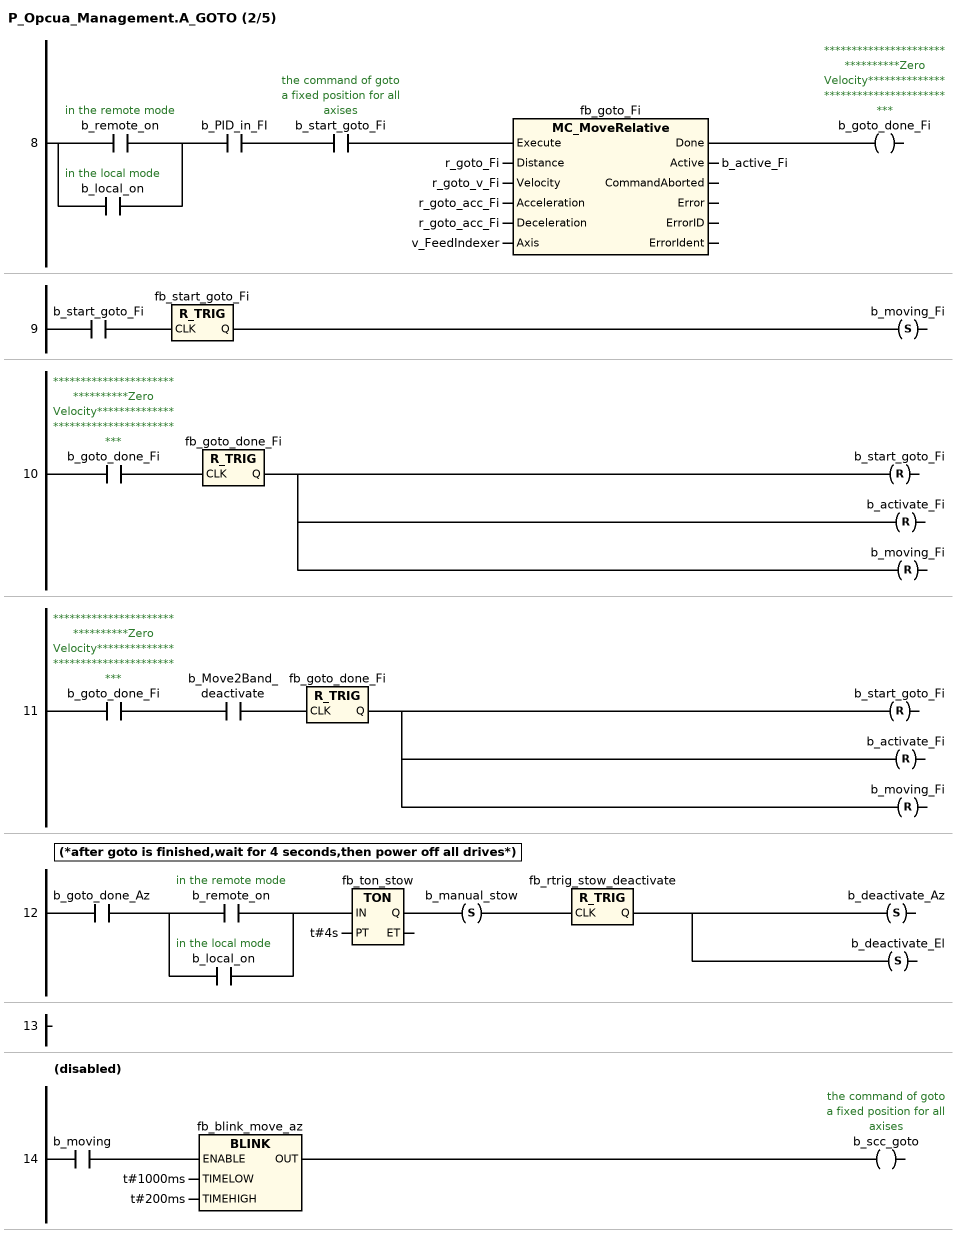
// NETWORK 8
//   b_remote_on: in the remote mode
//   b_local_on: in the local mode
//   b_start_goto_Fi: the command of goto a fixed position for all axises
//   r_goto_Fi: actual value of goto
//   v_FeedIndexer: Virtual axis "v_azimuth" with axis number 7
//   b_goto_done_Fi: ********************************Zero Velocity***************************************
fb_goto_Fi(
    Execute := (b_remote_on OR b_local_on) AND b_PID_in_FI AND b_start_goto_Fi,
    Distance := r_goto_Fi,
    Velocity := r_goto_v_Fi,
    Acceleration := r_goto_acc_Fi,
    Deceleration := r_goto_acc_Fi,
    Axis := v_FeedIndexer,
    Active => b_active_Fi); // MC_MoveRelative
b_goto_done_Fi := fb_goto_Fi.Done;

// NETWORK 9
fb_start_goto_Fi(CLK := b_start_goto_Fi); // R_TRIG
b_moving_Fi S= fb_start_goto_Fi.Q;

// NETWORK 10
//   b_goto_done_Fi: ********************************Zero Velocity***************************************
fb_goto_done_Fi(CLK := b_goto_done_Fi); // R_TRIG
b_start_goto_Fi R= fb_goto_done_Fi.Q;
b_activate_Fi R= fb_goto_done_Fi.Q;
b_moving_Fi R= fb_goto_done_Fi.Q;

// NETWORK 11
//   b_goto_done_Fi: ********************************Zero Velocity***************************************
fb_goto_done_Fi(CLK := b_goto_done_Fi AND b_Move2Band_deactivate); // R_TRIG
b_start_goto_Fi R= fb_goto_done_Fi.Q;
b_activate_Fi R= fb_goto_done_Fi.Q;
b_moving_Fi R= fb_goto_done_Fi.Q;

// NETWORK 12
//   fb_rtrig_stow_deactivate: the definition of rise trigger,The function block R_TRIG detects a rising edge.
//   fb_ton_stow: The function block Timer On Delay implements a turn-on delay
//   b_remote_on: in the remote mode
//   b_local_on: in the local mode
// label: (*after goto is finished,wait for 4 seconds,then power off all drives*)
fb_ton_stow(IN := b_goto_done_Az AND (b_remote_on OR b_local_on), PT := t#4s); // TON
b_manual_stow S= fb_ton_stow.Q;
fb_rtrig_stow_deactivate(CLK := fb_ton_stow.Q); // R_TRIG
b_deactivate_Az S= fb_rtrig_stow_deactivate.Q;
b_deactivate_El S= fb_rtrig_stow_deactivate.Q;

// NETWORK 13

// NETWORK 14 (disabled)
//   b_scc_goto: the command of goto a fixed position for all axises
// fb_blink_move_az(ENABLE := b_moving, TIMELOW := t#1000ms, TIMEHIGH := t#200ms); // BLINK
// b_scc_goto := fb_blink_move_az.OUT;

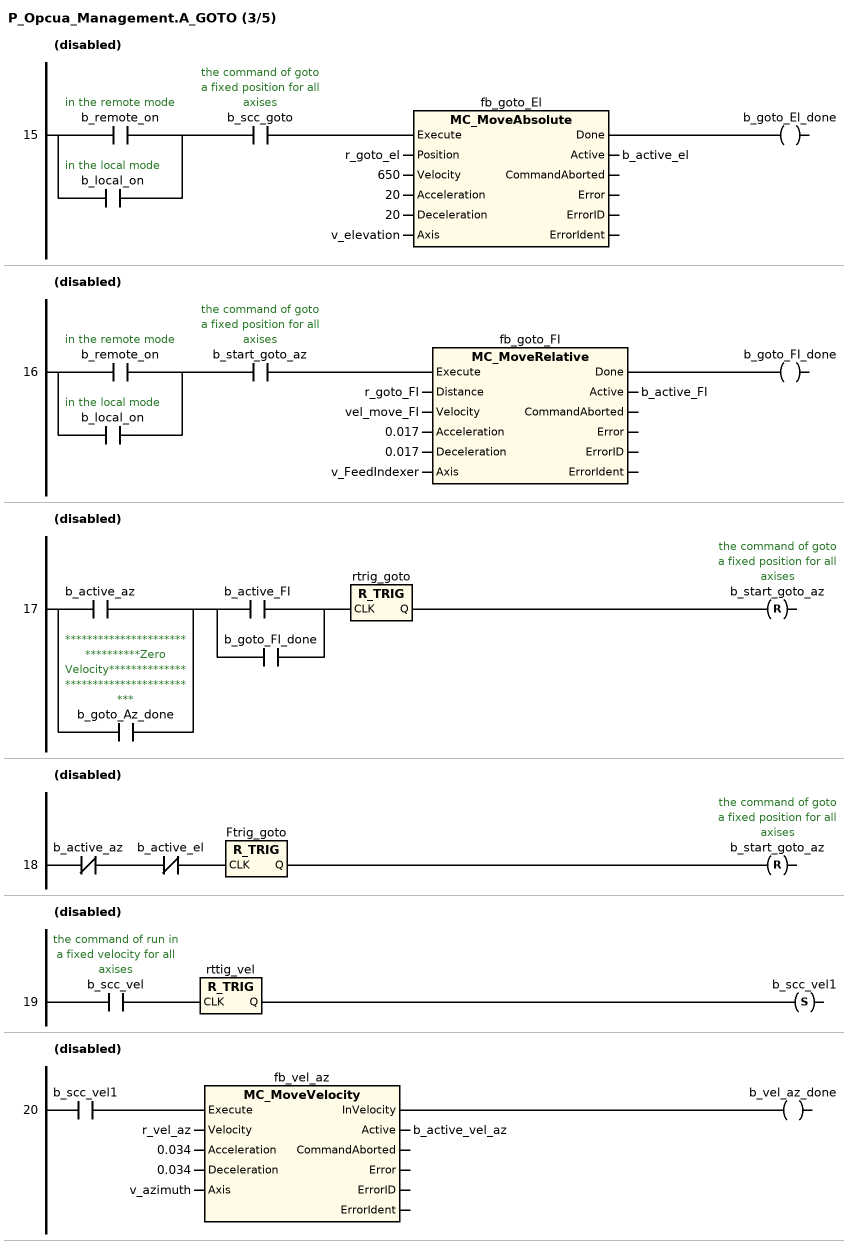
// NETWORK 15 (disabled)
//   b_remote_on: in the remote mode
//   b_local_on: in the local mode
//   b_scc_goto: the command of goto a fixed position for all axises
//   v_elevation: Virtual axis "v_elevation" with axis number 8
// fb_goto_El(
//     Execute := (b_remote_on OR b_local_on) AND b_scc_goto,
//     Position := r_goto_el,
//     Velocity := 650,
//     Acceleration := 20,
//     Deceleration := 20,
//     Axis := v_elevation,
//     Active => b_active_el); // MC_MoveAbsolute
// b_goto_El_done := fb_goto_El.Done;

// NETWORK 16 (disabled)
//   b_remote_on: in the remote mode
//   b_local_on: in the local mode
//   b_start_goto_az: the command of goto a fixed position for all axises
//   v_FeedIndexer: Virtual axis "v_polarization" with axis number 9
// fb_goto_FI(
//     Execute := (b_remote_on OR b_local_on) AND b_start_goto_az,
//     Distance := r_goto_FI,
//     Velocity := vel_move_FI,
//     Acceleration := 0.017,
//     Deceleration := 0.017,
//     Axis := v_FeedIndexer,
//     Active => b_active_FI); // MC_MoveRelative
// b_goto_FI_done := fb_goto_FI.Done;

// NETWORK 17 (disabled)
//   b_goto_Az_done: ********************************Zero Velocity***************************************
//   b_start_goto_az: the command of goto a fixed position for all axises
// rtrig_goto(CLK := (b_active_az OR b_goto_Az_done) AND (b_active_FI OR b_goto_FI_done)); // R_TRIG
// b_start_goto_az R= rtrig_goto.Q;

// NETWORK 18 (disabled)
//   b_start_goto_az: the command of goto a fixed position for all axises
// Ftrig_goto(CLK := NOT b_active_az AND NOT b_active_el); // R_TRIG
// b_start_goto_az R= Ftrig_goto.Q;

// NETWORK 19 (disabled)
//   b_scc_vel: the command of run in a fixed velocity for all axises
// rttig_vel(CLK := b_scc_vel); // R_TRIG
// b_scc_vel1 S= rttig_vel.Q;

// NETWORK 20 (disabled)
//   r_vel_az: ************vel*************
//   v_azimuth: Virtual axis "v_azimuth" with axis number 7
// fb_vel_az(
//     Execute := b_scc_vel1,
//     Velocity := r_vel_az,
//     Acceleration := 0.034,
//     Deceleration := 0.034,
//     Axis := v_azimuth,
//     Active => b_active_vel_az); // MC_MoveVelocity
// b_vel_az_done := fb_vel_az.InVelocity;

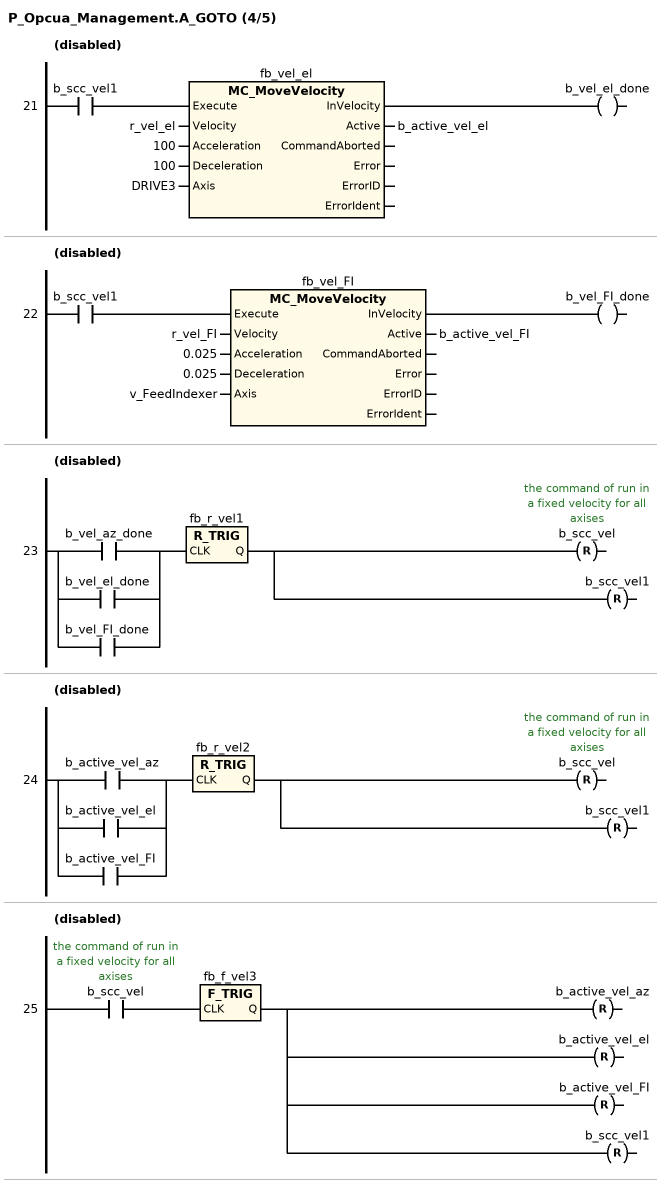
// NETWORK 21 (disabled)
//   DRIVE3: Virtual axis "v_elevation" with axis number 8
// fb_vel_el(
//     Execute := b_scc_vel1,
//     Velocity := r_vel_el,
//     Acceleration := 100,
//     Deceleration := 100,
//     Axis := DRIVE3,
//     Active => b_active_vel_el); // MC_MoveVelocity
// b_vel_el_done := fb_vel_el.InVelocity;

// NETWORK 22 (disabled)
//   v_FeedIndexer: Virtual axis "v_polarization" with axis number 9
// fb_vel_FI(
//     Execute := b_scc_vel1,
//     Velocity := r_vel_FI,
//     Acceleration := 0.025,
//     Deceleration := 0.025,
//     Axis := v_FeedIndexer,
//     Active => b_active_vel_FI); // MC_MoveVelocity
// b_vel_FI_done := fb_vel_FI.InVelocity;

// NETWORK 23 (disabled)
//   b_scc_vel: the command of run in a fixed velocity for all axises
// fb_r_vel1(CLK := b_vel_az_done OR b_vel_el_done OR b_vel_FI_done); // R_TRIG
// b_scc_vel R= fb_r_vel1.Q;
// b_scc_vel1 R= fb_r_vel1.Q;

// NETWORK 24 (disabled)
//   b_scc_vel: the command of run in a fixed velocity for all axises
// fb_r_vel2(CLK := b_active_vel_az OR b_active_vel_el OR b_active_vel_FI); // R_TRIG
// b_scc_vel R= fb_r_vel2.Q;
// b_scc_vel1 R= fb_r_vel2.Q;

// NETWORK 25 (disabled)
//   b_scc_vel: the command of run in a fixed velocity for all axises
// fb_f_vel3(CLK := b_scc_vel); // F_TRIG
// b_active_vel_az R= fb_f_vel3.Q;
// b_active_vel_el R= fb_f_vel3.Q;
// b_active_vel_FI R= fb_f_vel3.Q;
// b_scc_vel1 R= fb_f_vel3.Q;

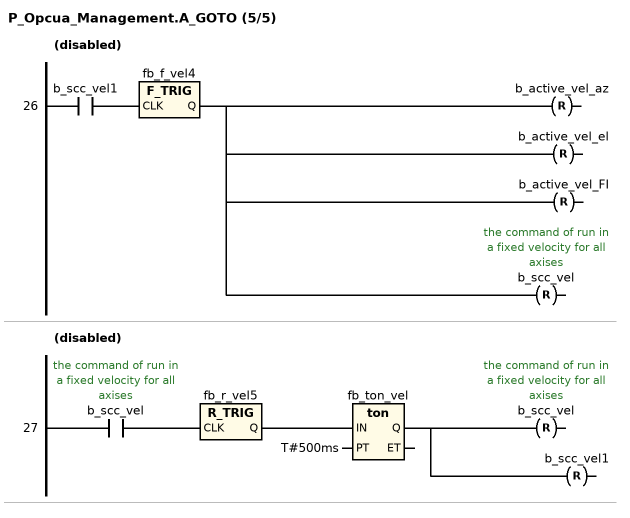
// NETWORK 26 (disabled)
//   b_scc_vel: the command of run in a fixed velocity for all axises
// fb_f_vel4(CLK := b_scc_vel1); // F_TRIG
// b_active_vel_az R= fb_f_vel4.Q;
// b_active_vel_el R= fb_f_vel4.Q;
// b_active_vel_FI R= fb_f_vel4.Q;
// b_scc_vel R= fb_f_vel4.Q;

// NETWORK 27 (disabled)
//   b_scc_vel: the command of run in a fixed velocity for all axises
// fb_r_vel5(CLK := b_scc_vel); // R_TRIG
// fb_ton_vel(IN := fb_r_vel5.Q, PT := T#500ms); // ton
// b_scc_vel R= fb_ton_vel.Q;
// b_scc_vel1 R= fb_ton_vel.Q;
END_ACTION

ACTION A_CLR_ERR:
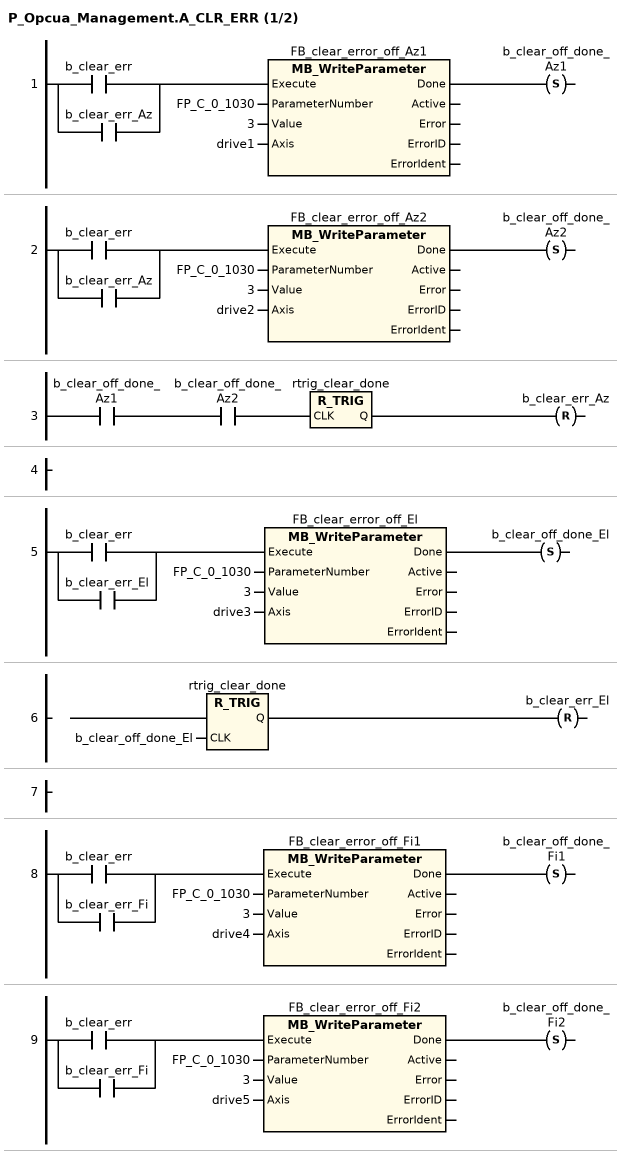
// NETWORK 1
//   FP_C_0_1030: Command: Clear all control errors
//   drive1: Real axis "Drive1" with axis number 1
FB_clear_error_off_Az1(
    Execute := b_clear_err OR b_clear_err_Az,
    ParameterNumber := FP_C_0_1030,
    Value := 3,
    Axis := drive1); // MB_WriteParameter
b_clear_off_done_Az1 S= FB_clear_error_off_Az1.Done;

// NETWORK 2
//   FP_C_0_1030: Command: Clear all control errors
//   drive2: Real axis "Drive1" with axis number 1
FB_clear_error_off_Az2(
    Execute := b_clear_err OR b_clear_err_Az,
    ParameterNumber := FP_C_0_1030,
    Value := 3,
    Axis := drive2); // MB_WriteParameter
b_clear_off_done_Az2 S= FB_clear_error_off_Az2.Done;

// NETWORK 3
rtrig_clear_done(CLK := b_clear_off_done_Az1 AND b_clear_off_done_Az2); // R_TRIG
b_clear_err_Az R= rtrig_clear_done.Q;

// NETWORK 4

// NETWORK 5
//   FP_C_0_1030: Command: Clear all control errors
//   drive3: Real axis "Drive1" with axis number 1
FB_clear_error_off_El(
    Execute := b_clear_err OR b_clear_err_El,
    ParameterNumber := FP_C_0_1030,
    Value := 3,
    Axis := drive3); // MB_WriteParameter
b_clear_off_done_El S= FB_clear_error_off_El.Done;

// NETWORK 6
rtrig_clear_done(CLK := b_clear_off_done_El); // R_TRIG
b_clear_err_El R= rtrig_clear_done.Q;

// NETWORK 7

// NETWORK 8
//   FP_C_0_1030: Command: Clear all control errors
//   drive4: Real axis "Drive1" with axis number 1
FB_clear_error_off_Fi1(
    Execute := b_clear_err OR b_clear_err_Fi,
    ParameterNumber := FP_C_0_1030,
    Value := 3,
    Axis := drive4); // MB_WriteParameter
b_clear_off_done_Fi1 S= FB_clear_error_off_Fi1.Done;

// NETWORK 9
//   FP_C_0_1030: Command: Clear all control errors
//   drive5: Real axis "Drive1" with axis number 1
FB_clear_error_off_Fi2(
    Execute := b_clear_err OR b_clear_err_Fi,
    ParameterNumber := FP_C_0_1030,
    Value := 3,
    Axis := drive5); // MB_WriteParameter
b_clear_off_done_Fi2 S= FB_clear_error_off_Fi2.Done;

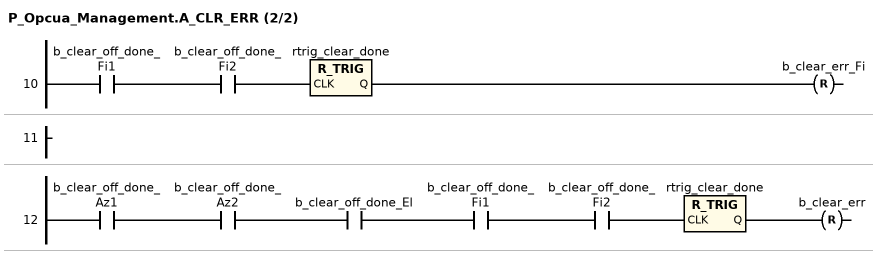
// NETWORK 10
rtrig_clear_done(CLK := b_clear_off_done_Fi1 AND b_clear_off_done_Fi2); // R_TRIG
b_clear_err_Fi R= rtrig_clear_done.Q;

// NETWORK 11

// NETWORK 12
rtrig_clear_done(CLK := b_clear_off_done_Az1 AND b_clear_off_done_Az2 AND b_clear_off_done_El AND b_clear_off_done_Fi1 AND b_clear_off_done_Fi2); // R_TRIG
b_clear_err R= rtrig_clear_done.Q;
END_ACTION

END_PROGRAM

// IndraMotionMlc1/Application/POUs/TCP/P_UDP_with_DAM
(*This program is built for UDP communication, receive the message from CSIRO,deal with the commands,and send the reply to CSIRO*)
PROGRAM P_UDP_with_DAM
VAR
(*<<<<<<<<<<<<<<<<<<<<<<<<<<<<<<<<<<<<<<<<<<<>>>>>>>>>>>>>>>>>>>>>>>>>>>>>>>>>>>>>*)
	b_receiving :BOOL;
	b_receiving_1 :BOOL;
	b_receiving_2 :BOOL;
	b_receiving_3 :BOOL;
	b_commanding: BOOL;
	b_commanding_1: BOOL;
	b_commanding_2: BOOL;
	b_commanding_3: BOOL;
	b_sending: BOOL;
	b_sending_1: BOOL;
	b_sending_2: BOOL;
	b_sending_3: BOOL;
	
(*<<<<<<<<<<<<<<<<<<<<<<<<<<<<<<<<<<<<<<<<<<<CONNECTION>>>>>>>>>>>>>>>>>>>>>>>>>>>>>>>>>>>>>*)
	UDPConnection_1: IL_UDPSocketAsync;
	UDPConnection_2: IL_UDPSocketAsync;
	UDPConnection_3: IL_UDPSocketAsync;
	b_Server_Enable: BOOL:=TRUE;(*the enable of IL_TCPConnectionAsync*)
	b_Server_Enable_1: BOOL:=TRUE;(*the enable of IL_TCPConnectionAsync*)
	b_Server_Enable_2: BOOL:=TRUE;(*the enable of IL_TCPConnectionAsync*)
	b_Server_Enable_3: BOOL:=TRUE;(*the enable of IL_TCPConnectionAsync*)
	di_Socket: DINT;(*the socket number*)
	di_Socket_1: DINT;(*the socket number*)
	di_Socket_2: DINT;(*the socket number*)
	di_Socket_3: DINT;(*the socket number*)
	strIP: STRING;
	b_Connection_done: BOOL;
	b_Connection_done_1: BOOL;
	b_Connection_done_2: BOOL;
	b_Connection_done_3: BOOL;
(*<<<<<<<<<<<<<<<<<<<<<<<<<<<<<<<<<<<<<<<<<<<RECEIVE>>>>>>>>>>>>>>>>>>>>>>>>>>>>>>>>>>>>>*)
	UDPRecv_1: IL_UDPRecvfromAsync;
	UDPRecv_2: IL_UDPRecvfromAsync;
	UDPRecv_3: IL_UDPRecvfromAsync;
	b_Recv_enable: BOOL;
	b_Recv_enable_1: BOOL;
	b_Recv_enable_2: BOOL;
	b_Recv_enable_3: BOOL;
	b_Recv_done: BOOL;
	b_Recv_done_1: BOOL;
	b_Recv_done_2: BOOL;
	b_Recv_done_3: BOOL;
	str_Recv: STRING(255);
	str_Recv_1: ARRAY [1..200] OF BYTE;
	str_Recv_2: ARRAY [1..200] OF BYTE;
	str_Recv_3: ARRAY [1..200] OF BYTE;
	//fb_crc16 : CRC16_MODBUS;
	di_ReceivedBytes: DINT;
	di_ReceivedBytes_1: DINT;
	di_ReceivedBytes_2: DINT;
	di_ReceivedBytes_3: DINT;
(*<<<<<<<<<<<<<<<<<<<<<<<<<<<<<<<<<<<<<<<<<<<<SEND>>>>>>>>>>>>>>>>>>>>>>>>>>>>>>>>>>>>>*)
	UDPSend_1: IL_UDPSendtoAsync;
	UDPSend_2: IL_UDPSendtoAsync;
	UDPSend_3: IL_UDPSendtoAsync;
	b_Send_enable: BOOL;
	b_Send_enable_1: BOOL;
	b_Send_enable_2: BOOL;
	b_Send_enable_3: BOOL;
	b_Send_done: BOOL;
	b_Send_done_1: BOOL;
	b_Send_done_2: BOOL;
	b_Send_done_3: BOOL;
	str_Send: STRING(1000);
	str_Send_1: ARRAY [1..8] OF BYTE;
	str_Send_2: ARRAY [1..8] OF BYTE;
	str_Send_3: ARRAY [1..8] OF BYTE;
	di_SentBytes: DINT;
	di_SentBytes_1: DINT;
	di_SentBytes_2: DINT;
	di_SentBytes_3: DINT;
	
	di_SentBytesLen_1: UINT;
	di_SentBytesLen_2: UINT;
	di_SentBytesLen_3: UINT;

(*add the function of close TCP function*)
	fb_tcp_close: IL_UDPCloseAsync;
	fb_udp_close_1: IL_UDPCloseAsync;
	fb_udp_close_2: IL_UDPCloseAsync;
	fb_udp_close_3: IL_UDPCloseAsync;
	B_TCP_close: BOOL;
	B_TCP_close_1: BOOL;
	B_TCP_close_2: BOOL;
	B_TCP_close_3: BOOL;
	b_TCP_close_done: BOOL;
	b_TCP_close_done_1: BOOL;
	b_TCP_close_done_2: BOOL;
	b_TCP_close_done_3: BOOL;
	b_Recv_active: BOOL;
	b_Recv_active_1: BOOL;
	b_Recv_active_2: BOOL;
	b_Recv_active_3: BOOL;
	i_counter_udp1:INT;
	i_counter_udp2:INT;
	i_counter_udp3:INT;

	str_concat: ARRAY[1..40] OF STRING(1000);(*数组及其类型的定义*)	
	str_concat_1: ARRAY[1..40] OF BYTE;(*数组及其类型的定义*)
	str_concat_2: ARRAY[1..40] OF BYTE;(*数组及其类型的定义*)
	str_concat_3: ARRAY[1..40] OF BYTE;(*数组及其类型的定义*)
	Counter: INT;
	bWaiting4Connection: BOOL;
	bWaiting4Connection_1: BOOL;
	bWaiting4Connection_2: BOOL;
	bWaiting4Connection_3: BOOL;
	bConnError: BOOL;
	bConnError_1: BOOL;
	bConnError_2: BOOL;
	bConnError_3: BOOL;
	diConnError: ERROR_CODE;
	diConnError_1: ERROR_CODE;
	diConnError_2: ERROR_CODE;
	diConnError_3: ERROR_CODE;
	ConnectError: ERROR_STRUCT;
	ConnectError_1: ERROR_STRUCT;
	ConnectError_2: ERROR_STRUCT;
	ConnectError_3: ERROR_STRUCT;
	i_counter_1s: INT:=0;	
	i_count:INT;
	
	reply_count: DINT;
	index: BYTE;
	
	dam1_data1 : LREAL;
	dam1_data2 : LREAL;
	dam1_data3 : LREAL;
	dam1_data4 : LREAL;
	dam1_data5 : LREAL;
	dam1_data6 : LREAL;
	dam1_data7 : LREAL;
	dam1_data8 : LREAL;
	dam1_data9 : LREAL;
	dam1_data10 : LREAL;
	dam1_data11 : LREAL;
	dam1_data12 : LREAL;
	

	
	dam3_data1 : REAL;
	dam3_data2 : REAL;
	dam3_data3 : REAL;
	dam3_data4 : REAL;
	dam3_data5 : REAL;
	dam3_data6 : REAL;
	dam3_data7 : REAL;
	dam3_data8 : REAL;
	dam3_data9 : REAL;
	dam3_data10 : REAL;
	dam3_data11 : REAL;
	dam3_data12 : REAL;
	dam3_data13 : REAL;
	dam3_data14 : REAL;
	dam3_data15 : REAL;
	dam3_data16 : REAL;
	dam3_data17 : REAL;
	dam3_data18 : REAL;
	dam3_data19 : REAL;
	dam3_data20 : REAL;
	dam3_data21 : REAL;
	dam3_data22 : REAL;
	dam3_data23 : REAL;
	dam3_data24 : REAL;
	dam3_data25 : REAL;
	dam3_data26 : REAL;
	dam3_data27 : REAL;
	dam3_data28 : REAL;
	fb_crc16_modbus: CRC16_MODBUS;
	
	a_phase_current : REAL;
	b_phase_current : REAL;
	c_phase_current : REAL;
	a_phase_voltage : REAL;
	b_phase_voltage : REAL;
	c_phase_voltage : REAL;
	ab_line_voltage : REAL;
	bc_line_voltage : REAL;
	ca_line_voltage : REAL;
	a_phase_activepower : REAL;
	b_phase_activepower : REAL;
	c_phase_activepower : REAL;
	a_phase_reactivepower : REAL;
	b_phase_reactivepower : REAL;
	c_phase_reactivepower : REAL;
	a_phase_apparentpower : REAL;
	b_phase_apparentpower : REAL;
	c_phase_apparentpower : REAL;
	a_phase_powerfactor : REAL;
	b_phase_powerfactor : REAL;
	c_phase_powerfactor : REAL;
	a_phase_frequency : REAL;
	b_phase_frequency : REAL;
	c_phase_frequency : REAL;
	total_activepower : REAL;
	total_reactivepower : REAL;
	total_apparentpower : REAL;
	total_powerfactor : REAL;
	
	
	X_Axis_Tile_Monitor : LREAL;
	Y_Axis_Tile_Monitor : LREAL;
	Temp_Tile_Monitor : LREAL;
	
	HumidEMISC_Outlet: LREAL;
END_VAR


reply_count:=reply_count+1;

IF reply_count < 0 OR reply_count >= 40 THEN	
	reply_count:=0;
END_IF

IF reply_count >= 0 AND reply_count < 10 THEN 
(*<<<<<<<<<<<<<<<<<<<<<<<<<<<<<concatenate STR_DAM1>>>>>>>>>>>>>>>>>>>>>>>>>>>>>>>>>>>>>>>>>>>>>>>>>>>>>>>*)
	str_concat_1[1] := 16#01;	//设备地址1
	str_concat_1[2] := 16#04;	//功能码
	str_concat_1[3] := 16#00;	//寄存器地址1
	str_concat_1[4] := 16#00;	//寄存器地址2
	str_concat_1[5] := 16#00;	//寄存器数量1
	str_concat_1[6] := 16#10;	//寄存器地址2
	fb_crc16_modbus(str_Message:= str_concat_1, str_Len:= 6, crc16=> );		//计算CRC校验
	str_concat_1[7] := WORD_TO_BYTE(fb_crc16_modbus.crc16 AND 16#00FF);
	str_concat_1[8] := WORD_TO_BYTE(SHR(fb_crc16_modbus.crc16,8) AND 16#00FF);
	FOR index:=1 TO 8 BY 1 DO
		str_send_1[index] := 16#00;
	END_FOR
	FOR index:=1 TO 8 BY 1 DO
		str_send_1[index] := str_concat_1[index];
	END_FOR
	di_SentBytesLen_1 := 8;
ELSIF reply_count >= 10 AND reply_count < 20 THEN
(*<<<<<<<<<<<<<<<<<<<<<<<<<<<<<concatenate STR_DAM2>>>>>>>>>>>>>>>>>>>>>>>>>>>>>>>>>>>>>>>>>>>>>>>>>>>>>>>*)
	str_concat_1[1] := 16#02;	//设备地址1
	str_concat_1[2] := 16#04;	//功能码
	str_concat_1[3] := 16#00;	//寄存器地址1
	str_concat_1[4] := 16#00;	//寄存器地址2
	str_concat_1[5] := 16#00;	//寄存器数量1
	str_concat_1[6] := 16#03;	//寄存器地址2
	fb_crc16_modbus(str_Message:= str_concat_1, str_Len:= 6, crc16=> );		//计算CRC校验
	str_concat_1[7] := WORD_TO_BYTE(fb_crc16_modbus.crc16 AND 16#00FF);
	str_concat_1[8] := WORD_TO_BYTE(SHR(fb_crc16_modbus.crc16,8) AND 16#00FF);
	FOR index:=1 TO 8 BY 1 DO
		str_send_1[index] := 16#00;
	END_FOR
	FOR index:=1 TO 8 BY 1 DO
		str_send_1[index] := str_concat_1[index];
	END_FOR
	di_SentBytesLen_1 := 8;
ELSIF reply_count >= 20 AND reply_count < 30 THEN
(*<<<<<<<<<<<<<<<<<<<<<<<<<<<<<concatenate STR_DAM2>>>>>>>>>>>>>>>>>>>>>>>>>>>>>>>>>>>>>>>>>>>>>>>>>>>>>>>*)
	str_concat_1[1] := 16#03;	//设备地址1
	str_concat_1[2] := 16#04;	//功能码
	str_concat_1[3] := 16#00;	//寄存器地址1
	str_concat_1[4] := 16#00;	//寄存器地址2
	str_concat_1[5] := 16#00;	//寄存器数量1
	str_concat_1[6] := 16#06;	//寄存器地址2
	fb_crc16_modbus(str_Message:= str_concat_1, str_Len:= 6, crc16=> );		//计算CRC校验
	str_concat_1[7] := WORD_TO_BYTE(fb_crc16_modbus.crc16 AND 16#00FF);
	str_concat_1[8] := WORD_TO_BYTE(SHR(fb_crc16_modbus.crc16,8) AND 16#00FF);
	FOR index:=1 TO 8 BY 1 DO
		str_send_1[index] := 16#00;
	END_FOR
	FOR index:=1 TO 8 BY 1 DO
		str_send_1[index] := str_concat_1[index];
	END_FOR
	di_SentBytesLen_1 := 8;
ELSE
(*<<<<<<<<<<<<<<<<<<<<<<<<<<<<<concatenate STR_DAM3>>>>>>>>>>>>>>>>>>>>>>>>>>>>>>>>>>>>>>>>>>>>>>>>>>>>>>>*)
	str_concat_1[1] := 16#03;	//设备地址1
	str_concat_1[2] := 16#04;	//功能码
	str_concat_1[3] := 16#00;	//寄存器地址1
	str_concat_1[4] := 16#27;	//寄存器地址2
	str_concat_1[5] := 16#00;	//寄存器数量1
	str_concat_1[6] := 16#0D;	//寄存器地址2
	fb_crc16_modbus(str_Message:= str_concat_1, str_Len:= 6, crc16=> );		//计算CRC校验
	str_concat_1[7] := WORD_TO_BYTE(fb_crc16_modbus.crc16 AND 16#00FF);
	str_concat_1[8] := WORD_TO_BYTE(SHR(fb_crc16_modbus.crc16,8) AND 16#00FF);
	FOR index:=1 TO 8 BY 1 DO
		str_send_1[index] := 16#00;
	END_FOR
	FOR index:=1 TO 8 BY 1 DO
		str_send_1[index] := str_concat_1[index];
	END_FOR	
	di_SentBytesLen_1 := 8;
END_IF
				
(*<<<<<<<<<<<<<<<<<<<<<<<<<<<if TCP is wrong,reset the TCP serve>>>>>>>>>>>>>>>>>>>>>>>>>>>>*)
IF UDPConnection_1.Error=TRUE OR UDPRecv_1.Error=TRUE OR UDPSend_1.Error=TRUE THEN
	b_Server_Enable_1:=FALSE;
	b_Recv_enable_1:=FALSE;
	b_Send_enable_1:=FALSE;
ELSE
	b_Server_Enable_1:=TRUE;
END_IF

IF UDPConnection_2.Error=TRUE OR UDPRecv_2.Error=TRUE OR UDPSend_2.Error=TRUE THEN
	b_Server_Enable_2:=FALSE;
	b_Recv_enable_2:=FALSE;
	b_Send_enable_2:=FALSE;
ELSE
	b_Server_Enable_2:=TRUE;
END_IF

P_UDP_with_DAM.Async_TCP();
P_UDP_with_DAM.A_RECV();
P_UDP_with_DAM.A_SEND();
(*<<<<<<<<<<<<<<<<<<<<<<<<<<<if TCP server is connected,a cycle is executed>>>>>>>>>>>>>>>>>>>>>>>>>>>>>>>>>>>>>>>>>>>>>*)
IF b_Connection_done_1=TRUE THEN
	IF  b_receiving_1=FALSE AND b_sending_1=FALSE AND b_Send_enable_1=FALSE THEN
		b_Send_enable_1:=TRUE;(*open send fuction*)
		P_UDP_with_DAM.A_SEND();
		b_sending_1:=TRUE;
	END_IF;
	
(*<<<<<<<<<<<<<<<<<<<<<<<<<<<send message>>>>>>>>>>>>>>>>>>>>>>>>>>>>>>>>>>>>>>>>>>>>>>>>>*)
	IF b_Send_done_1=TRUE AND b_sending_1=TRUE AND b_receiving_1=FALSE THEN
		b_Send_enable_1:=FALSE;
		P_UDP_with_DAM.A_SEND();
		b_sending_1:=FALSE;
		b_receiving_1:=TRUE;
		i_counter_udp1 := 0;
	END_IF;
	
(*<<<<<<<<<<<<<<<<<<<<<<<<<<<<<<<<<<<<<<<<<<<<<<<<<receive message>>>>>>>>>>>>>>>>>>>>>>>>>>>>>>>>>>>>>>>>>>>>>>>>>>>>>>>*)
	IF b_sending_1=FALSE AND b_receiving_1=TRUE THEN
		b_Recv_enable_1:=TRUE;
		P_UDP_with_DAM.A_RECV();
		i_counter_udp1 := i_counter_udp1 + 1;
	END_IF;
	
(*<<<<<<<<<<<<<<<<<<<<<<<<<<<<<<<<<<<<<<<<<<<<<<<<<not receive message>>>>>>>>>>>>>>>>>>>>>>>>>>>>>>>>>>>>>>>>>>>>>>>>>>>>>>>*)	
	IF b_sending_1=FALSE AND b_receiving_1=TRUE AND i_counter_udp1>10 THEN
		b_Recv_enable_1:=FALSE;
		b_receiving_1:=FALSE;
		i_counter_udp1 := 0;
	END_IF;
	
(*<<<<<<<<<<<<<<<<<<<<<<<<<<<recieveing message>>>>>>>>>>>>>>>>>>>>>>>>>>>>>>>>>>>>>>>>>>>>>>>>>*)
	IF b_Recv_done_1=TRUE AND b_receiving_1=TRUE THEN
		
		IF str_Recv_1[1] = 16#01 AND str_Recv_1[3] = 16#20 THEN
			
			HumidDriveCab := WORD_TO_LREAL(BYTE_TO_WORD(str_Recv_1[16]) * 256 + BYTE_TO_WORD(str_Recv_1[17])) / 65535 * 165 - 40;
			TempDriveCab := WORD_TO_LREAL(BYTE_TO_WORD(str_Recv_1[18]) * 256 + BYTE_TO_WORD(str_Recv_1[19])) / 65535 * 100;
			HumidPSC_Inlet := WORD_TO_LREAL(BYTE_TO_WORD(str_Recv_1[20]) * 256 + BYTE_TO_WORD(str_Recv_1[21])) / 65535 * 165 - 40;
			TempPSC_Inlet := WORD_TO_LREAL(BYTE_TO_WORD(str_Recv_1[22]) * 256 + BYTE_TO_WORD(str_Recv_1[23])) / 65535 * 100;
			HumidPSC_Outlet := WORD_TO_LREAL(BYTE_TO_WORD(str_Recv_1[24]) * 256 + BYTE_TO_WORD(str_Recv_1[25])) / 65535 * 165 - 40;
			TempPSC_Outlet := WORD_TO_LREAL(BYTE_TO_WORD(str_Recv_1[26]) * 256 + BYTE_TO_WORD(str_Recv_1[27])) / 65535 * 100;
			HumidEMISC_Outlet := WORD_TO_LREAL(BYTE_TO_WORD(str_Recv_1[28]) * 256 + BYTE_TO_WORD(str_Recv_1[29])) / 65535 * 100 - 20;
			TempEMISC_Outlet := WORD_TO_LREAL(BYTE_TO_WORD(str_Recv_1[30]) * 256 + BYTE_TO_WORD(str_Recv_1[31])) / 65535 * 100;
			dam1_data9 := WORD_TO_LREAL(BYTE_TO_WORD(str_Recv_1[32]) * 256 + BYTE_TO_WORD(str_Recv_1[33])) / 65535 * 100 - 20;
			dam1_data10 := WORD_TO_LREAL(BYTE_TO_WORD(str_Recv_1[34]) * 256 + BYTE_TO_WORD(str_Recv_1[35])) / 65535 * 100;
			
		ELSIF str_Recv_1[1] = 16#02 AND str_Recv_1[3] = 16#06 THEN
			
			Pedestal_temp_1 := WORD_TO_REAL(BYTE_TO_WORD(str_Recv_1[4]) * 256 + BYTE_TO_WORD(str_Recv_1[5])) / 65535 * 200 - 50;
			Pedestal_temp_2 := WORD_TO_REAL(BYTE_TO_WORD(str_Recv_1[6]) * 256 + BYTE_TO_WORD(str_Recv_1[7])) / 65535 * 200 - 50;
			Pedestal_temp_3 := WORD_TO_REAL(BYTE_TO_WORD(str_Recv_1[8]) * 256 + BYTE_TO_WORD(str_Recv_1[9])) / 65535 * 200 - 50;
			
		ELSIF str_Recv_1[1] = 16#03 AND str_Recv_1[3] =16#0C THEN
			
			CurrentPh1 := WORD_TO_LREAL(BYTE_TO_WORD(str_Recv_1[4]) * 256 + BYTE_TO_WORD(str_Recv_1[5])) / 65535 * 100;
			CurrentPh2 := WORD_TO_LREAL(BYTE_TO_WORD(str_Recv_1[6]) * 256 + BYTE_TO_WORD(str_Recv_1[7])) / 65535 * 100;
			CurrentPh3 := WORD_TO_LREAL(BYTE_TO_WORD(str_Recv_1[8]) * 256 + BYTE_TO_WORD(str_Recv_1[9])) / 65535 * 100;
			VoltagePh1 := WORD_TO_LREAL(BYTE_TO_WORD(str_Recv_1[10]) * 256 + BYTE_TO_WORD(str_Recv_1[11])) / 65535 * 800;
			VoltagePh2 := WORD_TO_LREAL(BYTE_TO_WORD(str_Recv_1[12]) * 256 + BYTE_TO_WORD(str_Recv_1[13])) / 65535 * 800;
			VoltagePh3 := WORD_TO_LREAL(BYTE_TO_WORD(str_Recv_1[14]) * 256 + BYTE_TO_WORD(str_Recv_1[15])) / 65535 * 800;
		
		ELSIF str_Recv_1[1] = 16#03 AND str_Recv_1[3] =16#1A THEN
		
			FrequencyPh1 := WORD_TO_LREAL(BYTE_TO_WORD(str_Recv_1[4]) * 256 + BYTE_TO_WORD(str_Recv_1[5])) / 65535 * 65;
			FrequencyPh2 := WORD_TO_LREAL(BYTE_TO_WORD(str_Recv_1[6]) * 256 + BYTE_TO_WORD(str_Recv_1[7])) / 65535 * 65;
			FrequencyPh3 := WORD_TO_LREAL(BYTE_TO_WORD(str_Recv_1[8]) * 256 + BYTE_TO_WORD(str_Recv_1[9])) / 65535 * 65;
		
			PowerFactor := WORD_TO_LREAL(BYTE_TO_WORD(str_Recv_1[28]) * 256 + BYTE_TO_WORD(str_Recv_1[29])) / 65535 * 2 - 1;
	
		END_IF;

		b_Recv_enable_1:=FALSE;
		P_UDP_with_DAM.A_RECV();
		b_receiving_1:=FALSE;
		i_counter_udp1 := 0;
	END_IF;
	
	IF b_Recv_done_1=TRUE  THEN
		b_Recv_enable_1:=FALSE;
		P_UDP_with_DAM.A_RECV();
	END_IF;
(*<<<<<<<<<<<<<<<<<<<<<<<<<<<<<<<<<<<<<<<<<<<<<If not conected,then reset receive and send function>>>>>>>>>>>>>>>>>>>>>>>>>>>>>>>>>>>>>>>>>>>>>>>>>>>>>>>*)
ELSE
	b_receiving_1:=FALSE;
	b_sending_1:=FALSE;
	b_Recv_enable_1:=FALSE;
	b_send_enable_1:=FALSE;
END_IF;

(*Tilt Sensor Receiving Data*)
IF b_Connection_done_2=TRUE THEN
	IF  b_receiving_2=FALSE AND b_sending_2=FALSE AND b_Recv_enable_2=FALSE THEN
		b_Recv_enable_2:=TRUE;(*open receive fuction*)
		P_UDP_with_DAM.A_RECV();
		b_receiving_2:=TRUE;
	END_IF;
	
	IF b_Recv_done_2=TRUE AND b_receiving_2=TRUE THEN
		Pointing.Status.TiltXRaw_mV_One:= WORD_TO_LREAL(BYTE_TO_WORD(str_Recv_2[22]) * 256 + BYTE_TO_WORD(str_Recv_2[23]));
		Pointing.Status.TiltYRaw_mV_One := WORD_TO_LREAL(BYTE_TO_WORD(str_Recv_2[24]) * 256 + BYTE_TO_WORD(str_Recv_2[25]));
		Pointing.Status.TiltTemp_One := WORD_TO_LREAL(BYTE_TO_WORD(str_Recv_2[26]) * 256 + BYTE_TO_WORD(str_Recv_2[27]));
		X_Axis_Tile_Monitor := WORD_TO_LREAL(BYTE_TO_WORD(str_Recv_2[30]) * 256 + BYTE_TO_WORD(str_Recv_2[31]));
		Y_Axis_Tile_Monitor := WORD_TO_LREAL(BYTE_TO_WORD(str_Recv_2[32]) * 256 + BYTE_TO_WORD(str_Recv_2[33]));
		Temp_Tile_Monitor := WORD_TO_LREAL(BYTE_TO_WORD(str_Recv_2[34]) * 256 + BYTE_TO_WORD(str_Recv_2[35]));
	
		b_Recv_enable_2:=FALSE;
		P_UDP_with_DAM.A_RECV();
		b_receiving_2:=FALSE;
	END_IF;
ELSE
	b_receiving_2:=FALSE;
	b_sending_2:=FALSE;
	b_Recv_enable_2:=FALSE;
	b_send_enable_2:=FALSE;
END_IF;

ACTION Async_TCP:
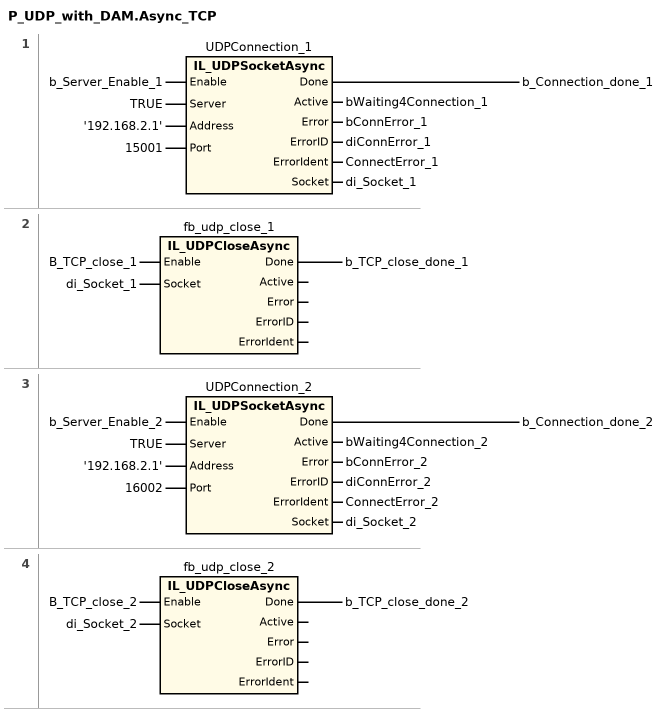
// NETWORK 1
UDPConnection_1(
    Enable := b_Server_Enable_1,
    Server := TRUE,
    Address := '192.168.2.1',
    Port := 15001,
    Active => bWaiting4Connection_1,
    Error => bConnError_1,
    ErrorID => diConnError_1,
    ErrorIdent => ConnectError_1,
    Socket => di_Socket_1); // IL_UDPSocketAsync
b_Connection_done_1 := UDPConnection_1.Done;

// NETWORK 2
fb_udp_close_1(Enable := B_TCP_close_1, Socket := di_Socket_1); // IL_UDPCloseAsync
b_TCP_close_done_1 := fb_udp_close_1.Done;

// NETWORK 3
UDPConnection_2(
    Enable := b_Server_Enable_2,
    Server := TRUE,
    Address := '192.168.2.1',
    Port := 16002,
    Active => bWaiting4Connection_2,
    Error => bConnError_2,
    ErrorID => diConnError_2,
    ErrorIdent => ConnectError_2,
    Socket => di_Socket_2); // IL_UDPSocketAsync
b_Connection_done_2 := UDPConnection_2.Done;

// NETWORK 4
fb_udp_close_2(Enable := B_TCP_close_2, Socket := di_Socket_2); // IL_UDPCloseAsync
b_TCP_close_done_2 := fb_udp_close_2.Done;
END_ACTION

ACTION A_RECV:
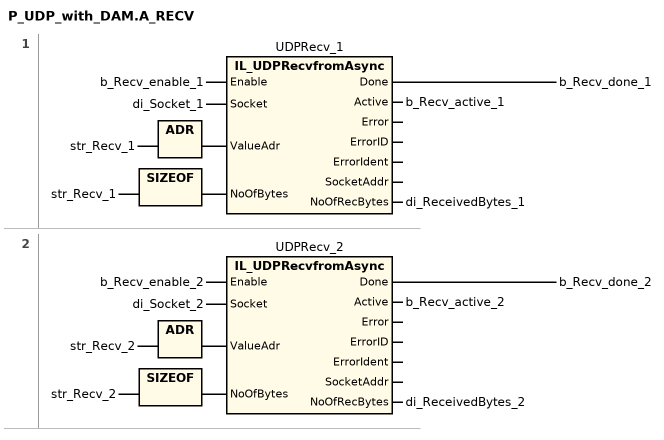
// NETWORK 1
UDPRecv_1(
    Enable := b_Recv_enable_1,
    Socket := di_Socket_1,
    ValueAdr := ADR(str_Recv_1),
    NoOfBytes := SIZEOF(str_Recv_1),
    Active => b_Recv_active_1,
    NoOfRecBytes => di_ReceivedBytes_1); // IL_UDPRecvfromAsync
b_Recv_done_1 := UDPRecv_1.Done;

// NETWORK 2
UDPRecv_2(
    Enable := b_Recv_enable_2,
    Socket := di_Socket_2,
    ValueAdr := ADR(str_Recv_2),
    NoOfBytes := SIZEOF(str_Recv_2),
    Active => b_Recv_active_2,
    NoOfRecBytes => di_ReceivedBytes_2); // IL_UDPRecvfromAsync
b_Recv_done_2 := UDPRecv_2.Done;
END_ACTION

ACTION A_SEND:
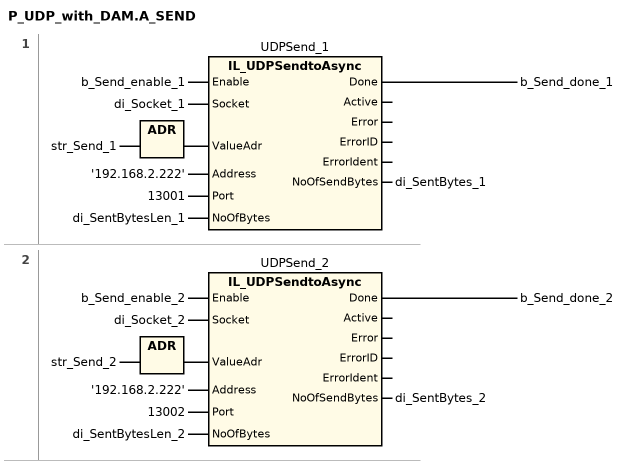
// NETWORK 1
UDPSend_1(
    Enable := b_Send_enable_1,
    Socket := di_Socket_1,
    ValueAdr := ADR(str_Send_1),
    Address := '192.168.2.222',
    Port := 13001,
    NoOfBytes := di_SentBytesLen_1,
    NoOfSendBytes => di_SentBytes_1); // IL_UDPSendtoAsync
b_Send_done_1 := UDPSend_1.Done;

// NETWORK 2
UDPSend_2(
    Enable := b_Send_enable_2,
    Socket := di_Socket_2,
    ValueAdr := ADR(str_Send_2),
    Address := '192.168.2.222',
    Port := 13002,
    NoOfBytes := di_SentBytesLen_2,
    NoOfSendBytes => di_SentBytes_2); // IL_UDPSendtoAsync
b_Send_done_2 := UDPSend_2.Done;
END_ACTION

END_PROGRAM

// IndraMotionMlc1/Application/POUs/TCP/Message/CRC16_MODBUS
FUNCTION_BLOCK CRC16_MODBUS
VAR_INPUT
	str_Message: ARRAY[1..40] OF BYTE;
	str_Len: BYTE;
END_VAR
VAR_OUTPUT
	crc16 : WORD;
END_VAR
VAR
	i : BYTE;
	j : BYTE;
	polynomial : WORD;
	curval : WORD;
	temp : WORD;
END_VAR


temp := 16#FFFF;
polynomial := 16#A001;
FOR i:=1 TO str_Len BY 1 DO
	curval := BYTE_TO_WORD(str_Message[i]);
	FOR j:=1 TO 8 BY 1 DO
		IF ((WORD_TO_BYTE(temp XOR curval) AND 16#01) = 16#01) THEN
			temp := (SHR(temp,1) XOR polynomial);
		ELSE
			temp := SHR(temp,1);			
		END_IF;
		curval := SHR(curval,1);
	END_FOR;
END_FOR;

crc16 := temp;

END_FUNCTION_BLOCK

// IndraMotionMlc1/Application/POUs/OPCUA/OPCUA_Node/P_Opcua_Tracking
{attribute 'linkalways'}
PROGRAM P_Opcua_Tracking
VAR_INPUT
	
	i_length: UINT;
	tai: ARRAY [1..1000] OF LREAL;
	Az: ARRAY [1..1000] OF LREAL;
	El: ARRAY [1..1000] OF LREAL;
	
END_VAR

VAR
	index: UINT; // Index used for addressing points in the tracking data arrays. 
	
	IL_LowPass_OnSource: IL_StateVariableType01;
	b_test: BOOL;
	
END_VAR


// Switch track on if the starttime has been reached
IF b_track_start AND (lr_track_start_time <= Time_cds.Status.TAIoffset) THEN 
	b_track_on:=1;
	b_track_start:=0;
END_IF

//IF i_length>0 THEN  // Load table into stack 
	
	
//END_IF

// Calculate whether the dish is on source. 

IF b_track_on THEN 
	IF  tracking.status.OnSourceDev <= Tracking.Status.OnSourceThreshold THEN 
		Management.Status.OnSource:=1;
	ELSE
		Management.Status.OnSource:=0;	
	END_IF
ELSE
	Management.Status.OnSource:=0;
END_IF

//Tracking.Status.act_statOffset_value_El  Updated in P_Track_cubic
//Tracking.Status.act_statOffset_value_Xel Updated in P_Track_cubic
//Tracking.Status.OnSourceDev              Updated in P_Track_cubic
//Tracking.Status.OnSourceThreshold        Updated in SetOnSourceThreshold
//Tracking.Status.p_desired_Az;            Updated in P_Track_cubic
//Tracking.Status.p_desired_El;            Updated in P_Track_cubic
//Tracking.Status.ThresholdTimePeriod      Updated in SetOnSourceThreshold
IF Management.Status.DscState=DscStatetype.Standby OR Management.Status.DscState=DscStatetype.Standstill OR Management.Status.DscState=DscStatetype.Slew OR Management.Status.DscState=DscStatetype.Track THEN 
	Tracking.Status.tr_initOk:=1;
ELSE 
	Tracking.Status.tr_initOk:=0;
END_IF

Tracking.Status.tr_obj_valid:= Tracking.TableStatus.pts_DataValid;
Tracking.Status.tr_selPoly:= 0;

IF Tracking.TableStatus.pts_DataValid THEN
	Tracking.Status.tr_TimeRemaining:= ABS(track_table[i_End].TAIoffset - track_table[i_Start].TAIoffset);
ELSE
	Tracking.Status.tr_TimeRemaining:=0;
END_IF

IF (track_table[i_End].TAIoffset)>(Time_cds.Status.TAIoffset+600) THEN  // Minimum of 10min track data available . 
	Tracking.Status.tr_valid:=1;
ELSE
	Tracking.Status.tr_valid:=0;
END_IF

Tracking.TableStatus.act_pt_act_index := INT_TO_UINT(i_Start);
Tracking.TableStatus.act_pt_end_index := INT_TO_UINT(i_End);
Tracking.TableStatus.act_pt_value_Az:= track_table[i_Start].Azimuth;
Tracking.TableStatus.act_pt_value_El:= track_table[i_Start].Elevation;
//Tracking.TableStatus.LastLoadMode; Updated in TrackloadTable
IF i_num_stack_left > 10 THEN
	Tracking.TableStatus.pts_Completed:=0; 
	ELSE
	Tracking.TableStatus.pts_Completed:=1;
END_IF
IF Tracking.TableStatus.pts_Completed THEN 
	Tracking.TableStatus.pts_DataValid:=0; // Once a track is finnished then there is no valid data to trck with. 
END_IF
Tracking.TableStatus.pts_Err:=0; 
//Tracking.TableStatus.pts_Interpol;  Updated in Track Start
Tracking.TableStatus.pts_InterpolError:=0;  // Don't have code for detecting interpolaor errors yet
Tracking.TableStatus.pts_Running:=b_track_on;
Tracking.TableStatus.pts_StartPos:=b_track_on;

IF i_num_stack_left<=60 AND i_num_stack_left >= 70 THEN
	Tracking.TableStatus.pts_TableAlmostFull:=1;
ELSE 
	Tracking.TableStatus.pts_TableAlmostFull:=0;
END_IF

P_Opcua_Tracking.A_Utils();

ACTION A_Utils:
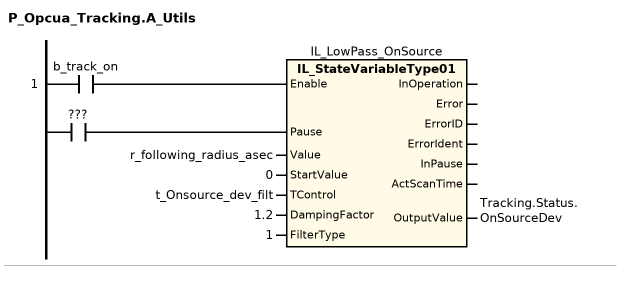
// NETWORK 1
IL_LowPass_OnSource(
    Enable := b_track_on,
    Value := r_following_radius_asec,
    StartValue := 0,
    TControl := t_Onsource_dev_filt,
    DampingFactor := 1.2,
    FilterType := 1,
    OutputValue => Tracking.Status.OnSourceDev); // IL_StateVariableType01
END_ACTION

END_PROGRAM

// IndraMotionMlc1/Application/POUs/OPCUA/OPCUA_Node/P_Opcua_Pointing
PROGRAM P_Opcua_Pointing
VAR
	TiltTemp_mV_1: LREAL;
	lr_one_x_off: LREAL;
	lr_one_y_off: LREAL;
	TiltTemp_mV_2: LREAL;
	lr_two_x_off: LREAL;
	lr_two_y_off: LREAL;
	IL_LowPass_Tilt_one_x: IL_StateVariableType01;
	IL_LowPass_Tilt_one_y: IL_StateVariableType01;
	IL_LowPass_Tilt_two_x: IL_StateVariableType01;
	IL_LowPass_Tilt_two_y: IL_StateVariableType01;
	t_one_x_filt_dt: TIME;
	t_one_y_filt_dt: TIME;
	t_two_x_filt_dt: TIME;
	t_two_y_filt_dt: TIME;
	b_tilt_filt_on: BOOL:= 1;
END_VAR

Pointing();
(*****Data*****)

(****************** Tilt Sensor **************************************)
// Tilt sensor one
Pointing.Status.TiltTemp_One := TiltTemp_mV_1*0.1;

lr_one_x_off:= (Pointing.TiltmeterParameters.One.x_zero+Pointing.TiltmeterParameters.One.x_zeroTC*Pointing.Status.TiltTemp_One)+
(Pointing.TiltmeterParameters.One.x_off+Pointing.TiltmeterParameters.One.x_offTC*Pointing.Status.TiltTemp_One);
lr_one_y_off:=(Pointing.TiltmeterParameters.One.y_zero+Pointing.TiltmeterParameters.One.y_zeroTC*Pointing.Status.TiltTemp_One)+
(Pointing.TiltmeterParameters.One.y_off+Pointing.TiltmeterParameters.One.y_offTC*Pointing.Status.TiltTemp_One);

Pointing.Status.TiltXArcsec_One:= Pointing.Status.TiltXRaw_mV_One*(Pointing.TiltmeterParameters.One.x_scale+Pointing.TiltmeterParameters.One.x_scaleTC*Pointing.Status.TiltTemp_One)+Pointing.TiltmeterParameters.One.x_off;
Pointing.Status.TiltYArcsec_One:= Pointing.Status.TiltYRaw_mV_One*(Pointing.TiltmeterParameters.One.y_scale+Pointing.TiltmeterParameters.One.y_scaleTC*Pointing.Status.TiltTemp_One)+Pointing.TiltmeterParameters.One.y_off;
t_one_x_filt_dt:= TO_TIME(Pointing.TiltmeterParameters.One.x_filt_dt*1000); //convert to milliseconds and TIME type.
t_one_y_filt_dt:= TO_TIME(Pointing.TiltmeterParameters.One.y_filt_dt*1000);

// Tilt Sensor Two
Pointing.Status.TiltTemp_Two := TiltTemp_mV_2*0.1;

lr_two_x_off:= (Pointing.TiltmeterParameters.Two.x_zero+Pointing.TiltmeterParameters.Two.x_zeroTC*Pointing.Status.TiltTemp_Two)+
(Pointing.TiltmeterParameters.Two.x_off+Pointing.TiltmeterParameters.Two.x_offTC*Pointing.Status.TiltTemp_Two);
lr_two_y_off:=(Pointing.TiltmeterParameters.Two.y_zero+Pointing.TiltmeterParameters.Two.y_zeroTC*Pointing.Status.TiltTemp_Two)+
(Pointing.TiltmeterParameters.Two.y_off+Pointing.TiltmeterParameters.Two.y_offTC*Pointing.Status.TiltTemp_Two);

Pointing.Status.TiltXArcsec_Two:= Pointing.Status.TiltXRaw_mV_Two*(Pointing.TiltmeterParameters.Two.x_scale+Pointing.TiltmeterParameters.Two.x_scaleTC*Pointing.Status.TiltTemp_Two)+Pointing.TiltmeterParameters.Two.x_off;
Pointing.Status.TiltYArcsec_Two:= Pointing.Status.TiltYRaw_mV_Two*(Pointing.TiltmeterParameters.Two.y_scale+Pointing.TiltmeterParameters.Two.y_scaleTC*Pointing.Status.TiltTemp_Two)+Pointing.TiltmeterParameters.Two.y_off;
t_two_x_filt_dt:= TO_TIME(Pointing.TiltmeterParameters.Two.x_filt_dt*1000); //convert to milliseconds and TIME type.
t_two_y_filt_dt:= TO_TIME(Pointing.TiltmeterParameters.Two.y_filt_dt*1000);

// Total point corrections

Pointing.Status.TotalPointCorr_Az:= Pointing.Status.StaticPmCorrVal_Az + Pointing.Status.TiltCorrVal_Az + Pointing.Status.AmbTempCorrVal_Az;
Pointing.Status.TotalPointCorr_El:= Pointing.Status.StaticPmCorrVal_El + Pointing.Status.TiltCorrVal_El + Pointing.Status.AmbTempCorrVal_El;

Pointing.Status.ActAmbTemp_East:= Pedestal_temp_1;  // These need to be checked
Pointing.Status.ActAmbTemp_South:= Pedestal_temp_2;;
Pointing.Status.ActAmbTemp_West:= Pedestal_temp_3;
//Pointing.Status.AmbTempCorrActive
//Pointing.Status.AmbTempCorrVal_Az
//Pointing.Status.AmbTempCorrVal_El
//Pointing.Status.BandForCorr
//Pointing.Status.StaticCorrActive
//Pointing.Status.StaticPmCorrVal_Az
//Pointing.Status.StaticPmCorrVal_El
//Pointing.Status.TiltCorrActive
//Pointing.Status.TiltCorrVal_Az
//Pointing.Status.TiltCorrVal_El
//Pointing.Status.TiltOne_On
//Pointing.Status.TiltTemp_One
//Pointing.Status.TiltTemp_Two
//Pointing.Status.TotalPointCorr_Az
//Pointing.Status.TotalPointCorr_El

ACTION A_Utils:
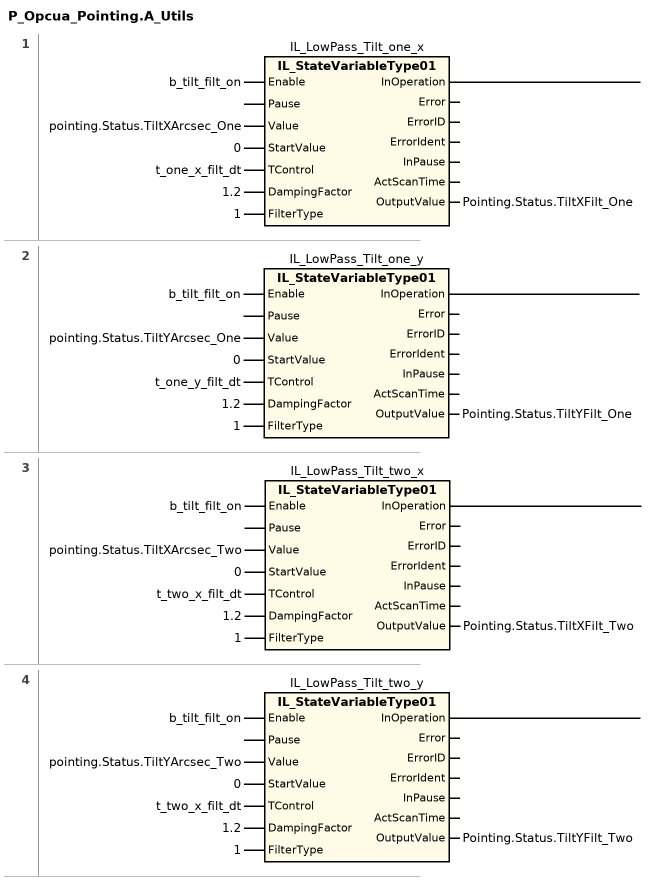
// NETWORK 1
IL_LowPass_Tilt_one_x(
    Enable := b_tilt_filt_on,
    Value := pointing.Status.TiltXArcsec_One,
    StartValue := 0,
    TControl := t_one_x_filt_dt,
    DampingFactor := 1.2,
    FilterType := 1,
    OutputValue => Pointing.Status.TiltXFilt_One); // IL_StateVariableType01

// NETWORK 2
IL_LowPass_Tilt_one_y(
    Enable := b_tilt_filt_on,
    Value := pointing.Status.TiltYArcsec_One,
    StartValue := 0,
    TControl := t_one_y_filt_dt,
    DampingFactor := 1.2,
    FilterType := 1,
    OutputValue => Pointing.Status.TiltYFilt_One); // IL_StateVariableType01

// NETWORK 3
IL_LowPass_Tilt_two_x(
    Enable := b_tilt_filt_on,
    Value := pointing.Status.TiltXArcsec_Two,
    StartValue := 0,
    TControl := t_two_x_filt_dt,
    DampingFactor := 1.2,
    FilterType := 1,
    OutputValue => Pointing.Status.TiltXFilt_Two); // IL_StateVariableType01

// NETWORK 4
IL_LowPass_Tilt_two_y(
    Enable := b_tilt_filt_on,
    Value := pointing.Status.TiltYArcsec_Two,
    StartValue := 0,
    TControl := t_two_x_filt_dt,
    DampingFactor := 1.2,
    FilterType := 1,
    OutputValue => Pointing.Status.TiltYFilt_Two); // IL_StateVariableType01
END_ACTION

END_PROGRAM

// IndraMotionMlc1/Application/POUs/Motion/Test_move
PROGRAM Test_move
VAR
	b_power: BOOL;
	b_enable_az1: BOOL;
	fb_enable_az1: MC_Power;
	b_enable_az1_done: BOOL;
	b_vel_az1: BOOL;
	fb_vel_az1: MC_MoveVelocity;
	vel_az1: REAL;
	b_enable_az2: BOOL;
	fb_enable_az2: MC_Power;
	b_enable_az2_done: BOOL;
	b_vel_az2: BOOL;
	vel_az2: REAL;
	fb_vel_az2: MC_MoveVelocity;
	b_enable_el1: BOOL;
	fb_enable_el1: MC_Power;
	b_enable_el1_done: BOOL;
	b_vel_el1: BOOL;
	vel_el1: REAL;
	fb_vel_el1: MC_MoveVelocity;
	b_vel_el2: BOOL;
	fb_vel_el2: MC_MoveVelocity;
	vel_el2: REAL;
	b_enable_el2: BOOL;
	fb_enable_el2: MC_Power;
	b_enable_FI1: BOOL;
	fb_enable_FI1: MC_Power;
	b_enable_el2_done: BOOL;
	b_enable_FI1_done: BOOL;
	b_vel_FI1: BOOL;
	fb_vel_FI1: MC_MoveVelocity;
	vel_FI1: REAL;
	b_enable_FI2: BOOL;
	fb_enable_FI2: MC_Power;
	b_enable_FI2_done: BOOL;
	b_vel_FI2: BOOL;
	vel_FI2: REAL;
	fb_vel_FI2: MC_MoveVelocity;
	b_torque_4: BOOL;
	b_torque_el2: BOOL;
	fb_torque_el2: MC_TorqueControl;
	b_torque_el2_done: BOOL;
	b_torque_az2: BOOL;
	fb_torque_az2: MC_TorqueControl;
	b_torque_az2_done: BOOL;
	fb_pos_az1: MC_MoveAbsolute;
	b_pos_az1: BOOL;
	pos_az1: REAL;
	b_stop_az: BOOL;
	fb_stop_AZ: MC_Stop;
	b_stop_el: BOOL;
	fb_stop_el: MC_Stop;
	b_pos_el1: BOOL;
	pos_el1: REAL;
	fb_pos_el1: MC_MoveAbsolute;
	b_pos_FI1: BOOL;
	pos_FI1: REAL;
	fb_pos_FI1: MC_MoveAbsolute;
	b_vel_1: BOOL;
	vel_1: REAL;
	fb_vel_1: MC_MoveVelocity;
	test_home_1: BOOL;
	fb_test_home: MB_Home;
	b_homeswitch_1: BOOL;
	b_torque_FI2: BOOL;
	fb_torque_FI2: MC_TorqueControl;
	b_torque_FI2_done: BOOL;
	b_touque_1: BOOL;
	fb_torque_az1: MC_TorqueControl;
	b_torque_az1_done: BOOL;
	torque_1: REAL;
	b_touque_3: BOOL;
	torque_3: REAL;
	fb_torque_el3: MC_TorqueControl;
END_VAR

(*IF r_pos_az>270.5 OR  r_pos_az<-270.5 THEN
			b_SCC_enable_on:=FALSE;
			b_SCC_enable_off:=TRUE; 
END_IF
*)




//axisdata[7].rActualPosition_i;
//test_move.power_move(); Commented out to prevent process using up resources.

ACTION power_move:
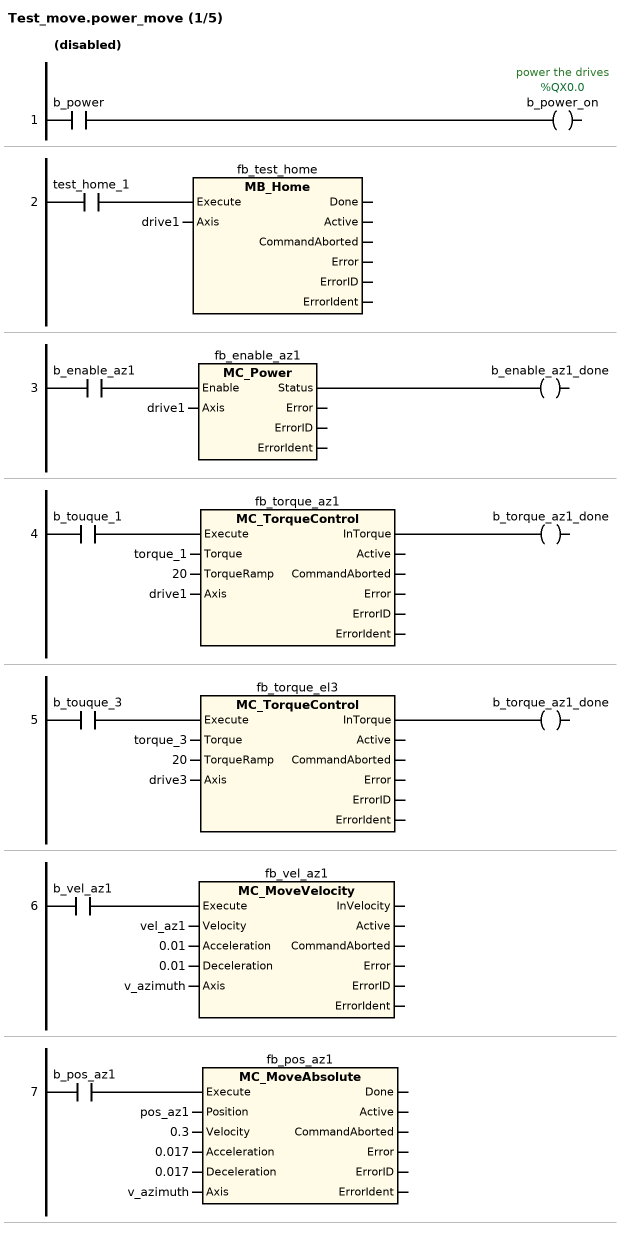
// NETWORK 1 (disabled)
//   b_power_on: power the drives | AT %QX0.0
// b_power_on := b_power;

// NETWORK 2
//   drive1: Real axis "Drive1" with axis number 1
fb_test_home(Execute := test_home_1, Axis := drive1); // MB_Home

// NETWORK 3
//   drive1: Real axis "Drive1" with axis number 1
fb_enable_az1(Enable := b_enable_az1, Axis := drive1); // MC_Power
b_enable_az1_done := fb_enable_az1.Status;

// NETWORK 4
//   drive1: Real axis "Drive4" with axis number 4
fb_torque_az1(Execute := b_touque_1, Torque := torque_1, TorqueRamp := 20, Axis := drive1); // MC_TorqueControl
b_torque_az1_done := fb_torque_az1.InTorque;

// NETWORK 5
//   drive3: Real axis "Drive4" with axis number 4
fb_torque_el3(Execute := b_touque_3, Torque := torque_3, TorqueRamp := 20, Axis := drive3); // MC_TorqueControl
b_torque_az1_done := fb_torque_el3.InTorque;

// NETWORK 6
//   v_azimuth: Virtual axis "v_azimuth" with axis number 7
fb_vel_az1(
    Execute := b_vel_az1,
    Velocity := vel_az1,
    Acceleration := 0.01,
    Deceleration := 0.01,
    Axis := v_azimuth); // MC_MoveVelocity

// NETWORK 7
//   v_azimuth: Virtual axis "v_azimuth" with axis number 7
fb_pos_az1(
    Execute := b_pos_az1,
    Position := pos_az1,
    Velocity := 0.3,
    Acceleration := 0.017,
    Deceleration := 0.017,
    Axis := v_azimuth); // MC_MoveAbsolute

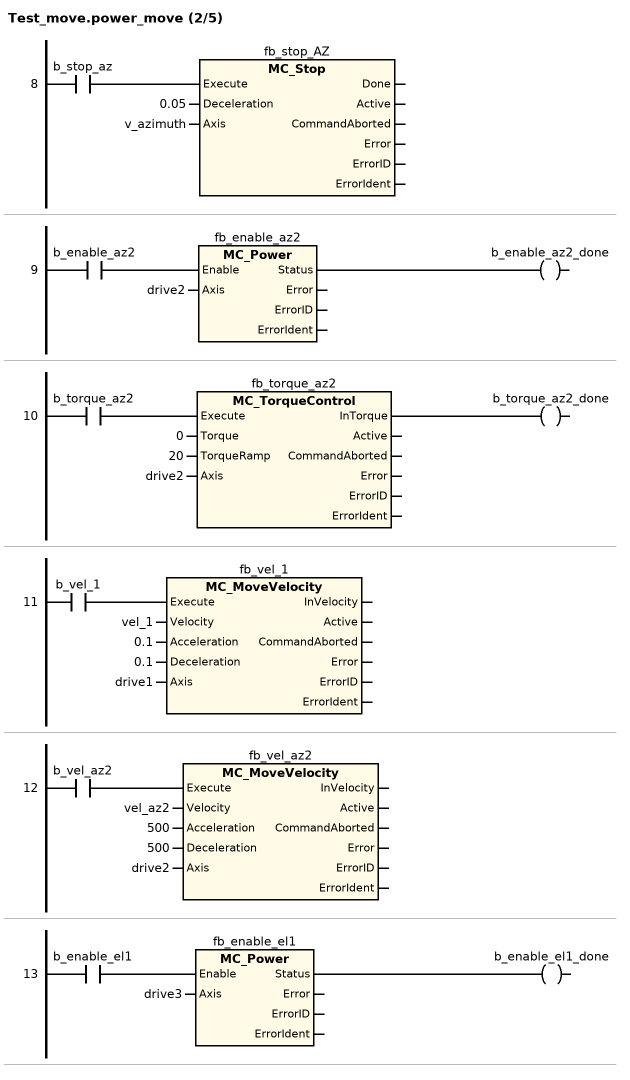
// NETWORK 8
//   v_azimuth: Virtual axis "v_azimuth" with axis number 7
fb_stop_AZ(Execute := b_stop_az, Deceleration := 0.05, Axis := v_azimuth); // MC_Stop

// NETWORK 9
//   drive2: Real axis "Drive2" with axis number 2
fb_enable_az2(Enable := b_enable_az2, Axis := drive2); // MC_Power
b_enable_az2_done := fb_enable_az2.Status;

// NETWORK 10
//   drive2: Real axis "Drive2" with axis number 2
fb_torque_az2(Execute := b_torque_az2, Torque := 0, TorqueRamp := 20, Axis := drive2); // MC_TorqueControl
b_torque_az2_done := fb_torque_az2.InTorque;

// NETWORK 11
//   drive1: Real axis "Drive1" with axis number 1
fb_vel_1(Execute := b_vel_1, Velocity := vel_1, Acceleration := 0.1, Deceleration := 0.1, Axis := drive1); // MC_MoveVelocity

// NETWORK 12
//   drive2: Real axis "Drive2" with axis number 2
fb_vel_az2(
    Execute := b_vel_az2,
    Velocity := vel_az2,
    Acceleration := 500,
    Deceleration := 500,
    Axis := drive2); // MC_MoveVelocity

// NETWORK 13
//   drive3: Real axis "Drive3" with axis number 3
fb_enable_el1(Enable := b_enable_el1, Axis := drive3); // MC_Power
b_enable_el1_done := fb_enable_el1.Status;

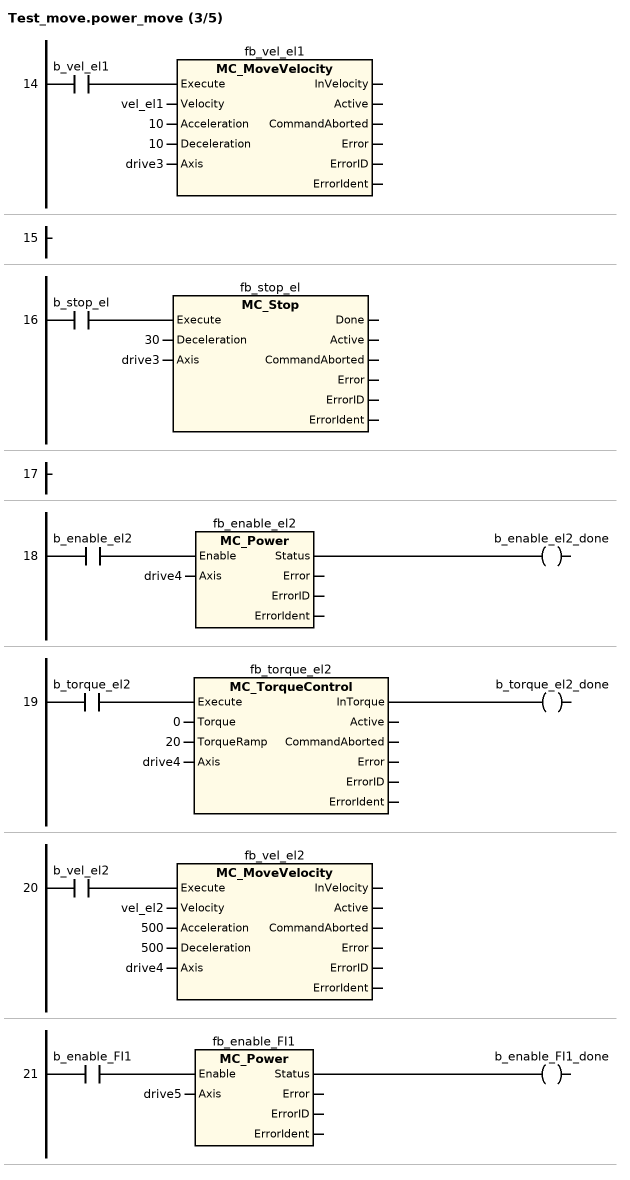
// NETWORK 14
//   drive3: Virtual axis "v_elevation" with axis number 8
fb_vel_el1(Execute := b_vel_el1, Velocity := vel_el1, Acceleration := 10, Deceleration := 10, Axis := drive3); // MC_MoveVelocity

// NETWORK 15

// NETWORK 16
//   drive3: Virtual axis "v_elevation" with axis number 8
fb_stop_el(Execute := b_stop_el, Deceleration := 30, Axis := drive3); // MC_Stop

// NETWORK 17

// NETWORK 18
//   drive4: Real axis "Drive4" with axis number 4
fb_enable_el2(Enable := b_enable_el2, Axis := drive4); // MC_Power
b_enable_el2_done := fb_enable_el2.Status;

// NETWORK 19
//   drive4: Real axis "Drive4" with axis number 4
fb_torque_el2(Execute := b_torque_el2, Torque := 0, TorqueRamp := 20, Axis := drive4); // MC_TorqueControl
b_torque_el2_done := fb_torque_el2.InTorque;

// NETWORK 20
//   drive4: Real axis "Drive4" with axis number 4
fb_vel_el2(
    Execute := b_vel_el2,
    Velocity := vel_el2,
    Acceleration := 500,
    Deceleration := 500,
    Axis := drive4); // MC_MoveVelocity

// NETWORK 21
//   drive5: Real axis "Drive5" with axis number 5
fb_enable_FI1(Enable := b_enable_FI1, Axis := drive5); // MC_Power
b_enable_FI1_done := fb_enable_FI1.Status;

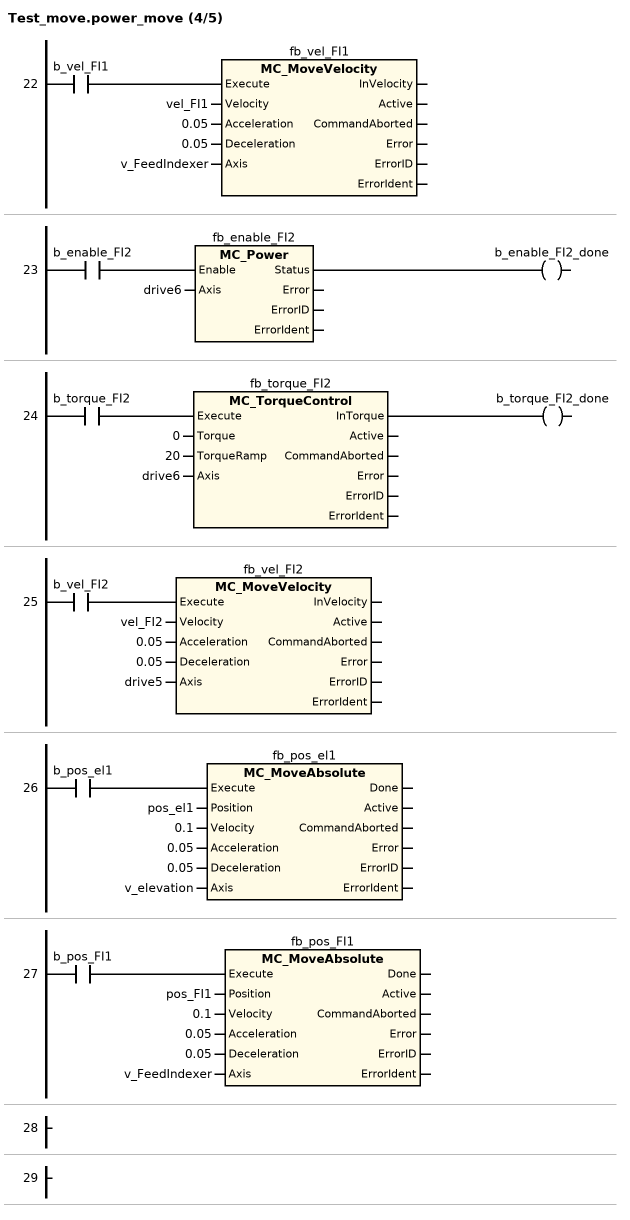
// NETWORK 22
//   v_FeedIndexer: Virtual axis "v_polarization" with axis number 9
fb_vel_FI1(
    Execute := b_vel_FI1,
    Velocity := vel_FI1,
    Acceleration := 0.05,
    Deceleration := 0.05,
    Axis := v_FeedIndexer); // MC_MoveVelocity

// NETWORK 23
//   drive6: Real axis "Drive6" with axis number 6
fb_enable_FI2(Enable := b_enable_FI2, Axis := drive6); // MC_Power
b_enable_FI2_done := fb_enable_FI2.Status;

// NETWORK 24
//   drive6: Real axis "Drive6" with axis number 6
fb_torque_FI2(Execute := b_torque_FI2, Torque := 0, TorqueRamp := 20, Axis := drive6); // MC_TorqueControl
b_torque_FI2_done := fb_torque_FI2.InTorque;

// NETWORK 25
//   drive5: Real axis "Drive5" with axis number 5
fb_vel_FI2(
    Execute := b_vel_FI2,
    Velocity := vel_FI2,
    Acceleration := 0.05,
    Deceleration := 0.05,
    Axis := drive5); // MC_MoveVelocity

// NETWORK 26
//   v_elevation: Virtual axis "v_elevation" with axis number 8
fb_pos_el1(
    Execute := b_pos_el1,
    Position := pos_el1,
    Velocity := 0.1,
    Acceleration := 0.05,
    Deceleration := 0.05,
    Axis := v_elevation); // MC_MoveAbsolute

// NETWORK 27
//   v_FeedIndexer: Virtual axis "v_polarization" with axis number 9
fb_pos_FI1(
    Execute := b_pos_FI1,
    Position := pos_FI1,
    Velocity := 0.1,
    Acceleration := 0.05,
    Deceleration := 0.05,
    Axis := v_FeedIndexer); // MC_MoveAbsolute

// NETWORK 28

// NETWORK 29

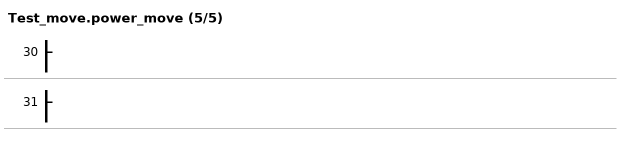
// NETWORK 30

// NETWORK 31
END_ACTION

END_PROGRAM

// IndraMotionMlc1/Application/POUs/Motion/PlcProg
PROGRAM PlcProg
VAR
	bVM_Enable: BOOL;
	rVM_Acc: REAL:=10.0;
	rVM_Dec: REAL:=10.0;
	rVM_Velocity: REAL:=3.0;
  rPhaseShift: REAL:=99.0;
	bVM_VelModeAck: BOOL;
	bVM_Standstill: BOOL;
	rVM_actVelocity: REAL;
END_VAR

//------------------------------------------------------------------------------------------------------
//--------------------- Call all required programs --> Imc and Axis Interface Update  ------------------  
//------------------------------------------------------------------------------------------------------
TE_AxisInterfaceType01Prog();
MB_ImcInterface();

IF TE_AxisInterfaceType01Prog.InitDone=FALSE THEN
	RETURN;
END_IF


//------------------------------------------------------------------------------------------------------
//----------------------------- Example for axis-access with AxisInterface ------------------------------  
//------------------------------------------------------------------------------------------------------

//----------------
// Axis-Command
//----------------
(*IF bRemoteOn_gb = FALSE THEN
 // arAxisCtrl_gb[MyVirtualAxis1.AxisNo].Admin._OpMode.b.MODE_VEL := bVM_Enable;
  IF bVM_Enable THEN
		arAxisCtrl_gb[MyVirtualAxis1.AxisNo].Admin._OpMode.en := ModeVel;
		arAxisCtrl_gb[MyVirtualAxis2.AxisNo].Admin._OpMode.en := ModeSyncPhase;
	ELSE
		arAxisCtrl_gb[MyVirtualAxis1.AxisNo].Admin._OpMode.en := ModeAb;
		arAxisCtrl_gb[MyVirtualAxis2.AxisNo].Admin._OpMode.en := ModeAb;
	END_IF
  arAxisCtrl_gb[MyVirtualAxis1.AxisNo].VelMode.Acceleration := rVM_Acc;
  arAxisCtrl_gb[MyVirtualAxis1.AxisNo].VelMode.Deceleration := rVM_Dec;
  arAxisCtrl_gb[MyVirtualAxis1.AxisNo].VelMode.Velocity := rVM_Velocity;
  arAxisCtrl_gb[MyVirtualAxis2.AxisNo].SyncMode.Master := MyVirtualAxis1;
  arAxisCtrl_gb[MyVirtualAxis2.AxisNo].SyncMode.PhaseShift := rPhaseShift;
END_IF
//----------------
// Axis-Status 
//----------------
bVM_VelModeAck := arAxisStatus_gb[MyVirtualAxis1.AxisNo].Admin.MODE_VEL;
IF (arAxisStatus_gb[MyVirtualAxis1.AxisNo].Admin.Active = TRUE) THEN
  // Pointer access only when axis is available -> avoid exceptions
  bVM_Standstill := arAxisStatus_gb[MyVirtualAxis1.AxisNo].PtrAxisData^.Axis_Standstill;
  rVM_actVelocity := arAxisStatus_gb[MyVirtualAxis1.AxisNo].PtrAxisData^.rActualVelocity_i;
END_IF
// Axis information can be evualated directly from AxisData-Array (same information at PtrAxisData^)
// AxisData[VM_Axis.AxisNo].Axis_Standstill;
// AxisData[VM_Axis.AxisNo].rActualVelocity_i;
*)

END_PROGRAM

// IndraMotionMlc1/Application/AxisInterface/TE_AxisInterfaceType01Prog
PROGRAM TE_AxisInterfaceType01Prog
(*#############################################################################################
  #############################################################################################  

   General Header   
  ---------------------------------------------------------------------------------------------  
   Shortdescription       : Cyclic execution of the Axis-Interface (POS, VEL and SYNC mode)
   Version                : see Version Function
   Name                   : DC-IA/EAM4 (KG)
   Date                   : see Version Function
   Company                : see Version Function
   Target                 : see Version Function
   Functional description : This program executes cyclic the axis interface FB for all axes.
                            The execution time of the axis interface FB is measured.
   Handling specials      : The global arrays of the axis-interface must be named arAxisCtrl_gb[]
                            and arAxisStatus_gb[]
  ---------------------------------------------------------------------------------------------  
    
   Additional Header   
  ---------------------------------------------------------------------------------------------  
  #############################################################################################  
  #############################################################################################*)
(*
                                     ******************
                                     *   DISCLAIMER   *
                                     ******************
   It is acknowledged that with regard to these software programs and program modules free of
   charge, Bosch Rexroth's usually practised, in-house test and release procedures have not 
   been accomplished. These software programs and program modules free of charge serve only as
   an example for possible applications.  They are intended as a help in order to obtain addi-
   tional experience regarding function, operation, performance and capacity of a maybe later 
   issued series release. Therefore Bosch Rexroth disclaims any liability and rejects to assume
   responsibility that these software programs or program modules, including any information 
   and data stored in those programs, are suitable for any intended use or that these programs
   will work without errors in any combination with the data processing environment. Providing
   you with these software programs shall neither constitute a claim for technical support nor
   for any other remedy for defects. Any claims for damages of any nature and for any legal
   reason arising from installing or using these software programs or program modules are ex-
   cluded, unless these damages was caused by Bosch Rexroth`s statutory representatives or em-
   ployees by wilful misconduct or by gross negligence or liability is compulsory in accordance
   with the German product liability law. In any case Bosch Rexroth`s liability for any conse-
   quential or incidental damages such as, but not limited to loss of profit, loss of pro-
   duction or loss of data is excluded.      
*)
(*---------------------------------------------------------------------------------------------*)
VAR_INPUT
  ClearError: BOOL;		// clear internal errors of the program
END_VAR
VAR_OUTPUT
  InitDone: BOOL;		// Init is done, AxisInterface is ready to operate
  Error: BOOL;			// internal error of the program
  ErrorID: ERROR_CODE;
  ErrorIdent: ERROR_STRUCT;
END_VAR
VAR CONSTANT
   STATE_FIRST_INIT       : UINT := 0;
   STATE_WAIT_FOR_PHASE2  : UINT := 1;
   STATE_INIT_P2          : UINT := 2;
   STATE_WAIT_FOR_PHASE3  : UINT := 3;
   STATE_INIT_P3          : UINT := 4;
   STATE_WAIT_FOR_PHASE4  : UINT := 5;
   STATE_WAIT_FOR_NOT_P4  : UINT := 6;
   STATE_PRG_ERROR        : UINT := 9;
   
   dwADD1_STATE_MACHINE_ERROR: DWORD := 16#00000006;
   dwADD2_STATE_MACHINE_ERROR: DWORD := 16#00000000;
   
END_VAR
VAR
    fbAxisInitAllAxis: TE_AxisInitAllAxisType01; //  basic init of arAxisCtrl structure 

    uiState                 : UINT := STATE_FIRST_INIT; // statemachine
	  // Flag that the inputs of the FB are set
	  bInitReferencesDone: BOOL; 
  
    fbAxis                    : ARRAY [1..uiMAX_AXIS_INDEX] OF TE_AxisInterface;
	  uiLoop                    : UINT := 1;
    uiAxisIdx                 : UINT; // axis index for the list without gaps
	  // time measurement
    udiStartTime              : UDINT;
    udiStopTime               : UDINT;
	  udiActCycleTime           : UDINT;
    stCyclesTime              : TE_PLC_CYCLES_TIME;
END_VAR

// -------------------------------------------------------------------------------- 
// state-machine: do the warmstart initialisation everytime we reach SERCOS phase 4 
// -------------------------------------------------------------------------------- 
CASE uiState OF

  STATE_FIRST_INIT:
    // ---------------------------------------------------------------------------------
    // Step: Done only once when PLC program starts.           
    // ---------------------------------------------------------------------------------
   	FOR uiLoop := 1 TO uiMAX_AXIS_INDEX DO
		 	fbAxis[uiLoop].mInitExtension(uiLoop);
		END_FOR
		bInitReferencesDone := TRUE; // Inputs are set, FB can be called	
    uiState := STATE_WAIT_FOR_PHASE2;
  
  STATE_WAIT_FOR_PHASE2:
    // --------------------------------------------------------------------------------- 
    // Step: Wait for SERCOS phase P2;                                                   
    // Done cyclic when we are in phases < 2                                             
    // --------------------------------------------------------------------------------- 
    IF (ImcStatus.Admin.ModeStatus_P2 = TRUE) THEN
      uiState := STATE_INIT_P2;
      InitDone := FALSE;      
		ELSIF( (ImcStatus.Admin.PwrUpModeAck = TRUE) AND (ImcStatus.Admin._OpModeAck > IMC_MODE_STATUS_P2) ) THEN
  	// E.g. PL program download in P4, go directly to P4
      uiState := STATE_INIT_P3;
      InitDone := FALSE;      
    END_IF
	
  STATE_INIT_P2:
    // --------------------------------------------------------------------------------- 
    // Step: Action actInitWarmStart. Done when reaching parameter mode.                 
    // --------------------------------------------------------------------------------- 
    actInitWarmStart();

  STATE_WAIT_FOR_PHASE3:
    // --------------------------------------------------------------------------------- 
    // Step: Wait for SERCOS phase P3;                 
    // Start Init once when reaching CP3                                   
    // ---------------------------------------------------------------------------------
    IF( ImcStatus.Admin._OpModeAck >= IMC_MODE_STATUS_P3 ) THEN
      uiState := STATE_INIT_P3;
      InitDone := FALSE;      
    END_IF


  STATE_INIT_P3:
    // --------------------------------------------------------------------------------- 
    // Step: Action actInitWarmStart. Done when reaching CP3                 
    // --------------------------------------------------------------------------------- 
    actInitWarmStart();

  STATE_WAIT_FOR_PHASE4:
    // --------------------------------------------------------------------------------- 
    // Step: Wait for SERCOS phase P4;                                                   
    // ---------------------------------------------------------------------------------
    IF( ImcStatus.Admin.ModeStatus_BB = TRUE ) THEN
      uiState := STATE_WAIT_FOR_NOT_P4;
    END_IF
    // Falling back into CP2 ? Return 
    IF (ImcStatus.Admin.ModeStatus_P2 = TRUE) THEN
      uiState := STATE_INIT_P2;
      InitDone := FALSE;      
    END_IF

  STATE_WAIT_FOR_NOT_P4:
    // --------------------------------------------------------------------------------- 
    // Step: Check SECROS phase changes from P4                                          
    // Done cyclic when we are in phase 4                                                
    // --------------------------------------------------------------------------------- 

    // Check if we have left phase 4 
    IF( (ImcStatus.Admin.ModeStatus_BB = FALSE) OR (InitDone = FALSE) ) THEN
      // We have left phase 4 -> re-init the axis interface 
      uiState := STATE_WAIT_FOR_PHASE4;
    END_IF
	
  STATE_PRG_ERROR:
    IF ClearError = TRUE THEN
      // clear error information
      Error := FALSE;
      InitDone := FALSE; // enforce a new init 
      uiState := STATE_WAIT_FOR_PHASE4;
    END_IF
	
  ELSE
	// -------------------------------------------- 
    // DEFAULT case -> Signal error !!!                      
    // -------------------------------------------- 
    Error := TRUE;
    // set error information
    ErrorID := STATE_MACHINE_ERROR;
    ErrorIdent.Table := F_RELATED_TABLE;
	  ErrorIdent.Additional1 := dwADD1_STATE_MACHINE_ERROR;
	  ErrorIdent.Additional2 := dwADD2_STATE_MACHINE_ERROR;
    uiState := STATE_PRG_ERROR; 

END_CASE

udiStartTime := IL_HighResTimeTick(TRUE); // latch starting time 

IF (InitDone AND bInitReferencesDone) THEN
  FOR uiLoop := 1 TO uiNofAxis_gb DO
    uiAxisIdx := arAxisIdx_gb[uiLoop];
		// comment the next line for performance optimisation, but then do no online-change!!!
		fbAxis[uiAxisIdx].mInitExtension(uiAxisIdx); // set inputs always to avoid online change problems  
    fbAxis[uiAxisIdx]( ); // call FB, inputs are already set....
  END_FOR
END_IF  

udiStopTime := IL_HighResTimeTick(TRUE); // latch end time 

// calculate actual runtime and store MIN and MAX 
udiActCycleTime := IL_HighResTimeDiff(udiStartTime,udiStopTime);

stCyclesTime.udiActualTime := udiActCycleTime;

IF (stCyclesTime.udiMaximumTime < udiActCycleTime) THEN
  stCyclesTime.udiMaximumTime := udiActCycleTime;
END_IF

IF (stCyclesTime.udiMinimumTime > udiActCycleTime) THEN
  stCyclestime.udiMinimumTime := udiActCycleTime;
END_IF

ACTION actInitWarmStart:
// --------------------------------------------------------------------------------- 
// Action actInitWarmStart: Done when reaching parameter mode (P2)                   
// and again when reaching operating mode (phase 4)             	             
// --------------------------------------------------------------------------------- 

// ############################################ 
// Step: Basic Init of arAxisCtrl_gb for all axes  
// ############################################ 
fbAxisInitAllAxis(
  Execute:= TRUE,
  ReadModuloValue:=TRUE,
  EnableCyclicScanning:=TRUE );

IF(fbAxisInitAllAxis.Error = TRUE) THEN
  // -------------------------------------------- 
  // Signal error !!!                      
  // -------------------------------------------- 
  Error := TRUE;
  // copy error information
  ErrorID := fbAxisInitAllAxis.ErrorID;
  ErrorIdent := fbAxisInitAllAxis.ErrorIdent;
  // reset FB 
  fbAxisinitAllAxis( Execute := FALSE );
  // go to error state
  uiState := STATE_PRG_ERROR; 
  
ELSIF(fbAxisInitAllAxis.Done = TRUE) THEN
  // -------------------------------------------- 
  // Signal init is finished                      
  // -------------------------------------------- 
  InitDone := TRUE; // Init is finished 
  // reset FB 
  fbAxisinitAllAxis( Execute := FALSE );
  

  // ---------------------------------------------------------------------------------
  // End of this state by increasing uiState (call from STATE_INIT_P2 or STATE_INIT_P4)                                          
  // ---------------------------------------------------------------------------------
  uiState := uiState + 1;
END_IF
END_ACTION

END_PROGRAM

// IndraMotionMlc1/Application/AxisInterface/TE_AxisInitAllAxisType01
(* Initialisation of the Axis-Interface (POS, VEL and SYNC mode)
  #############################################################################################
  #############################################################################################  

   General Header   
  ---------------------------------------------------------------------------------------------  
   Shortdescription       : Initialisation of the Axis-Interface (POS, VEL and SYNC mode)
   Version                : see Version Function
   Name                   : Dc-IA/EAM (KG,PoVa)
   Date                   : see Version Function
   Company                : see Version Function  
   Target                 : see Version Function
   Functional description : This functionblocks initialises the data structures for the
                            axis interface. All available axes (C-0-0484) are activated.
   Handling specials      : The global arrays of the axis-interface must be named arAxisCtrl_gb[]
                            and arAxisStatus_gb[]. The variables for the axis list without gaps 
                            must be named arAxisIdx_gb and uiNofAxis_gb. 
  ---------------------------------------------------------------------------------------------  
    
   Additional Header   
     The following structure elements are set by this function block:
      arAxisCtrl_gb[].Admin._OpMode.en = ModeAB
      arAxisCtrl_gb[].Admin.ClearError = FALSE      
      arAxisCtrl_gb[].Admin.LockInputChanges = FALSE       
      arAxisCtrl_gb[].Admin.SetAbsRef = FALSE      
      arAxisCtrl_gb[].Admin.Axis.CntrlNo = LOCAL_CNTRL;
      arAxisCtrl_gb[].Admin.Axis.AxisNo = AXIS_1 .. AXIS_n
      arAxisCtrl_gb[].PosMode.Adjust.Enable = FALSE       
      arAxisCtrl_gb[].VelMode.Adjust.Enable = FALSE       
      arAxisCtrl_gb[].SyncMode.AdjCamShaftDist.Enable = FALSE       
      arAxisCtrl_gb[].SyncMode.AdjFineadjust.Enable = FALSE         
      arAxisCtrl_gb[].SyncMode.AdjPhaseOffset.Enable = FALSE        
      arAxisCtrl_gb[].Comment = A-0-0002

      arAxisStatus_gb[].Active = TRUE for active axis ( C-0-0484 )
      arAxisStatus_gb[].Admin.AxisFeatures = set with value of A-0-0004 for all axis

    Only when ReadModuloValue = TRUE and the axis is rotatoric:
      arAxisCtrl_gb[iAxisNo].PosMode.Adjust.ModuloValue = A-0-0045
      arAxisCtrl_gb[iAxisNo].SyncMode.AdjPhaseOffset.ModuloValue = A-0-045
      arAxisCtrl_gb[iAxisNo].VelMode.Adjust.ModuloValue = 0
      arAxisCtrl_gb[iAxisNo].SyncMode.AdjCamShaftDist.ModuloValue = 0
      arAxisCtrl_gb[iAxisNo].SyncMode.AdjFineadjust.ModuloValue = 0

  ---------------------------------------------------------------------------------------------  
     
     
     
  ---------------------------------------------------------------------------------------------  

  #############################################################################################  
  #############################################################################################*)
(*
                                     ******************
                                     *   DISCLAIMER   *
                                     ******************
   It is acknowledged that with regard to these software programs and program modules free of
   charge, Bosch Rexroth's usually practised, in-house test and release procedures have not 
   been accomplished. These software programs and program modules free of charge serve only as
   an example for possible applications.  They are intended as a help in order to obtain addi-
   tional experience regarding function, operation, performance and capacity of a maybe later 
   issued series release. Therefore Bosch Rexroth disclaims any liability and rejects to assume
   responsibility that these software programs or program modules, including any information 
   and data stored in those programs, are suitable for any intended use or that these programs
   will work without errors in any combination with the data processing environment. Providing
   you with these software programs shall neither constitute a claim for technical support nor
   for any other remedy for defects. Any claims for damages of any nature and for any legal
   reason arising from installing or using these software programs or program modules are ex-
   cluded, unless these damages was caused by Bosch Rexroth`s statutory representatives or em-
   ployees by wilful misconduct or by gross negligence or liability is compulsory in accordance
   with the German product liability law. In any case Bosch Rexroth`s liability for any conse-
   quential or incidental damages such as, but not limited to loss of profit, loss of pro-
   duction or loss of data is excluded.      
*)
(*---------------------------------------------------------------------------------------------*)

FUNCTION_BLOCK TE_AxisInitAllAxisType01

VAR_INPUT
    Execute         : BOOL;            (* start execution with rising edge *)
    ReadModuloValue : BOOL := TRUE;    (* Read parameters A59 and A45 and write the modulo value
                                          for rotatoric axis to the adjustment structure of PosMode
                                          SyncMode.AdjPhaseOffset and set modulo value to 0 for all
                                          other adjusted values. Activate before "Execute" *)
    EnableCyclicScanning : BOOL := TRUE; (* Enable the cyclic check and transmission of changed
                                            inputs for the actual operating mode
                                            - relevant for the values in AxisCtrl with 
                                              "Note: cyclic checked AND transmitted on change" *)
END_VAR

VAR_OUTPUT
    {attribute 'analysis' := '-27'} // disable static code analysis rule 27, check of same names 
    Done        : BOOL := FALSE;       (* Is SET when FB has finished operation *)
    Active      : BOOL := FALSE;       (* Is SET when FB is active (not in idle mode) *)
    {attribute 'analysis' := '-27'} // disable static code analysis rule 27, check of same names 
    Error       : BOOL := FALSE;       (* ErrorFlag *)
    ErrorID     : ERROR_CODE;          (* Error identification, Errorcode *)
    ErrorIdent  : ERROR_STRUCT;        (* Error identification *)
END_VAR

VAR
    bOldExecute         : BOOL := FALSE;
    uiState             : UINT := 0;
    stDummyAxis         : AXIS_REF;
    arBuffer            : ARRAY [1..(MB_MAX_AXIS_NUMBER*2)] OF INT;
    fbReadListParaC484  : MB_ReadListParameter;
    uiAxisNo            : UINT   := 1;
    Axis                : AXIS_REF;
    fbAxisInitType01    : MB_AxisInitType01;
    uiLoop              : UINT;
END_VAR

VAR CONSTANT
   STATE_DO_NOTHING             : UINT := 0;
   STATE_READ_C484              : UINT := 1;
   STATE_CHK_AXIS               : UINT := 2;
   STATE_START_INIT             : UINT := 3;
	 STATE_ERROR									: UINT := 99;
END_VAR

(* Detect rising edge *)
IF( (Execute = TRUE) AND (bOldExecute = FALSE) ) THEN
     uiState := STATE_READ_C484;
END_IF

CASE uiState OF

    STATE_DO_NOTHING:
      IF( Execute = FALSE ) THEN
        (* RESET everything *)
        Done    := FALSE;
        Active  := FALSE;
        Error   := FALSE;
        uiAxisNo := 1;
      END_IF;

    STATE_READ_C484:
      (* ############################################### *)
      (* Step: Read C-0-0484 "Axes configuration list"   *)
      (* ############################################### *)

      fbReadListParaC484(
        Execute           := TRUE,
        ParameterNumber   := FP_C_0_0484,
        NoOfBytes         := SIZEOF(arBuffer),
        ValueAdr          := ADR(arBuffer),
        Axis              := stDummyAxis);

      IF ( fbReadListParaC484.Done = TRUE ) THEN
        (* reset FB *)
        fbReadListParaC484(
          Execute    := FALSE,
          Axis       := stDummyAxis);
        uiState := STATE_CHK_AXIS;
        uiAxisNo := 1;
        // reset list of all axes
        FOR uiLoop:=1 TO uiMAX_AXIS_INDEX DO
          arAxisIdx_gb[uiLoop] := 0;
				END_FOR
        uiNofAxis_gb := 0; // reset global axis counter 
      ELSIF ( fbReadListParaC484.Error = TRUE ) THEN
				Error := TRUE;
        ErrorID := fbReadListParaC484.ErrorID;
				ErrorIdent := fbReadListParaC484.ErrorIdent;
        (* reset FB *)
        fbReadListParaC484(
          Execute    := FALSE,
          Axis       := stDummyAxis);
        uiState := STATE_ERROR;
      END_IF

  STATE_CHK_AXIS:
    (* ############################################ *)
    (* Step: Check all configured axis              *)
    (* ############################################ *)
    IF ( uiAxisNo <= uiMAX_AXIS_INDEX ) THEN
      (* activate, when axis type not equal 0 *)
      IF ( arBuffer[2*uiAxisNo - 1] <> 0 ) THEN
        uiState      := STATE_START_INIT;
        Axis.AxisNo := UINT_TO_INT(uiAxisNo);
        Axis.CntrlNo := LOCAL_CNTRL;
        uiNofAxis_gb:=uiNofAxis_gb+1; // increase axes counter
        arAxisIdx_gb[uiNofAxis_gb] := uiAxisNo; // store the index in the lagless list 
      ELSE
        uiAxisNo := uiAxisNo + 1;
      END_IF

    ELSE
      Done    := TRUE;
      Active  := FALSE;
      uiState := STATE_DO_NOTHING;
    END_IF

  STATE_START_INIT:
    (* ############################################ *)
    (* Step: Initialize all configured axis         *)
    (* ############################################ *)

    (* call FB ML_AxisInitType01 -> initialize the axis *)
    fbAxisInitType01(
      Execute              := TRUE,
      ReadModuloValue      := ReadModuloValue,
      EnableCyclicScanning := EnableCyclicScanning,
      AdminCtrl            := arAxisCtrl_gb[uiAxisNo].Admin,
      PosModeCtrl          := arAxisCtrl_gb[uiAxisNo].PosMode,
      VelModeCtrl          := arAxisCtrl_gb[uiAxisNo].VelMode,
      SyncModeCtrl         := arAxisCtrl_gb[uiAxisNo].SyncMode,
      AxisDataPtrStatus    := arAxisStatus_gb[uiAxisNo].PtrAxisData,
      AdminStatus          := arAxisStatus_gb[uiAxisNo].Admin,
      DiagStatus           := arAxisStatus_gb[uiAxisNo].Diag,
      Axis                 := Axis);
    IF ( fbAxisInitType01.Error = TRUE ) THEN
      Error      := fbAxisInitType01.Error;
      ErrorID    := fbAxisInitType01.ErrorID;
      ErrorIdent := fbAxisInitType01.ErrorIdent;
 		  uiState    := STATE_ERROR;
    ELSIF ( fbAxisInitType01.Done = TRUE ) THEN
      (* restart ML_AxisInitType01 *)
      fbAxisInitType01(
        Execute            := FALSE,
        AdminCtrl          := arAxisCtrl_gb[uiAxisNo].Admin,
        PosModeCtrl        := arAxisCtrl_gb[uiAxisNo].PosMode,
        VelModeCtrl        := arAxisCtrl_gb[uiAxisNo].VelMode,
        SyncModeCtrl       := arAxisCtrl_gb[uiAxisNo].SyncMode,
        AxisDataPtrStatus  := arAxisStatus_gb[uiAxisNo].PtrAxisData,
        AdminStatus        := arAxisStatus_gb[uiAxisNo].Admin,
        DiagStatus         := arAxisStatus_gb[uiAxisNo].Diag,
        Axis               := Axis);
      (* check next axis *)
      uiAxisNo := uiAxisNo + 1;
      (* proceed with STATE_DO -> check next configured axis *)
      uiState := STATE_CHK_AXIS;

    END_IF

  STATE_ERROR:
        Active  := FALSE;
        Error   := TRUE;
        IF( (Execute = FALSE) AND (bOldExecute = TRUE) ) THEN
          uiState := STATE_DO_NOTHING;
        END_IF
				
	ELSE
	  ErrorID    := STATE_MACHINE_ERROR;
		ErrorIdent.Table := USER1_TABLE;
		ErrorIdent.Additional1 := uiState;
    ErrorIdent.Additional2 := 0;
		uiState    := STATE_ERROR;  
END_CASE

(* Edge detection *)
bOldExecute := Execute;

END_FUNCTION_BLOCK

// IndraMotionMlc1/Application/AxisInterface/TE_AxisInterface
// Online changes in declaration of axis-interface need too much time -> not allowed because risk of F5180006 
// InhibitOnlineChange = 0x1000000 has to be set decimal 16777216
{attribute 'signature_flag' := '16777216'} 
FUNCTION_BLOCK TE_AxisInterface EXTENDS MB_AxisInterfaceType01
(*#############################################################################################
  #############################################################################################  

  General Header   
  ---------------------------------------------------------------------------------------------  
  Shortdescription       : AxisInterface Example 
  Version                : see Version Function
  Name                   : DCC/EAM (DT/KG)
  Date                   : see Version Function
  Company                : see Version Function
  Target                 : see Version Function
  Functional description : Location in order to extend the AxisInterface functionality
  Handling specials      : This functionality is automatically assigned to the task the approriate
                           axis is assigned to
  ---------------------------------------------------------------------------------------------  
  
  Additional Header   
  ---------------------------------------------------------------------------------------------  

  ---------------------------------------------------------------------------------------------  

